	// ====== Axis enable =====	
		bCmdEnableAxis 		: BOOL 	:= FALSE; // Command to enable the axis (External)
		bInternalEnable		: BOOL 	:= FALSE; // internal enable command (turns off after set time, and on at new motion command
		bDelayedEnable		: BOOL 	:= false; // Delayed enable signal for motion commands
		TonMotionEnable		: TON 			; // Timer on for motion command enable
		TofIntAxisEnable	: TOF  			; // Timer off for internal axis enable 
	// ===== Safe commands =====
		bCmdSafeStop	: BOOL ;
	// Motion commands 
		fbMcPower 			: MC_Power		;		// FB for enable and override
		fbMcReset 			: MC_Reset		;		// FB to reset axis
		fbSoeReset			: FB_SoEReset	; 		// FB to reset axis hardware
		fbMcHome			: MC_Home		;		// Fb to home Axis
		fbMcStop 			: MC_Stop		;		// FB to stop axis
		fbMcHalt			: MC_Halt		;		// FB to halt axis
		fbMcJog				: MC_Jog		;		// FB to Jog axis
		fbMcMoveVelocity	: MC_MoveVelocity;		// FB to move with specified velocity until Next command is given
	(* PtoP Motion move commands are in arrays so multiple commands can be stacked *) 
		fbMCMoveRelative	: ARRAY [0..1] OF MC_MoveRelative	;		// FB to move relative
		fbMcMoveAbsolute	: ARRAY [0..1] OF MC_MoveAbsolute	;		// FB to move axis (velocity movement)
		
	// Parameters 
		stMParMaxAcc : Udt_Parameter := (fMaximum := 999999, fMinimum := 0, fValue := 0)	; // Parameter for maximum acceleration
		stMParMaxDec : Udt_Parameter := (fMaximum := 999999, fMinimum := 0, fValue := 0)	; // Parameter for maximum Deceleration
		stMparMaxVelo: Udt_Parameter := (fMaximum := 999999, fMinimum := 0, fValue := 0)	; // Parameter for maximum velocity
		
	// Device feedback
		nActVelocity AT%I* : INT ; // actual speed of the motor
		nActPosition AT%I* : UDINT ; // Actual position of the motor

	// ===== Function execute triggers =====
		bExec_Reset			: BOOL := FALSE; // Execute reset
		bExec_Halt			: BOOL := FALSE; // Execute hold
		bExec_Home			: BOOL := FALSE; // Execute Home
		bExec_JogPositive	: BOOL := FALSE; // Execute Jog in positive direction
		bExec_JogNegative	: BOOL := FALSE; // Execute Jog in negative direction
		bExec_MoveVelocity	: BOOL := FALSE; // Execute move velocity
		arExec_MoveRelative	: ARRAY [0..1] OF BOOL ; // Execute move relative
		arExec_MoveAbs		: ARRAY [0..1] OF BOOL ; // Execute move absolute reverse
		

END_VAR

// Call base function
SUPER^();

// ==== Check if axis is initiated =====
IF NOT bInitOk THEN 
	RETURN ; 
END_IF

// ===== Execute safe functions =====
	ExecSafeFunctions(); 

// ==== Execute organizational functions =====
	ExecEnable();

// ==== execute motion functions =====
	CallMotionFunctions();

METHOD PRIVATE CallMotionFunctions : BOOL
VAR_INPUT
END_VAR
// ===== Check if safe to move =====
	IF bCmdSafeStop OR NOT bDelayedEnable THEN 
		RETURN ;
	END_IF

// ===== Homing functions =====
	ExecHome		(); 

// ===== Motion standstil commands =====
	ExecHalt		();

// ===== Motion move functions
	ExecJog			(); 
	ExecMoveAbsolute();
	ExecMoveRelative();
	ExecMoveVelocity();
END_METHOD

METHOD PUBLIC CmdHalt : BOOL
VAR_INPUT
	fDeceleration 	: LREAL := 0 ; // command deceleration
	mcBuffermode	: MC_BufferMode ; // Buffermode defines how the previous command is executed.
END_VAR
// Set command to true 
bExec_Halt 		:= TRUE ;
bInternalEnable	:= TRUE ;

// copy parameters
fbMcHalt.Deceleration	:= fDeceleration;
fbMcHalt.BufferMode		:= mcBuffermode	;

// Set feedback output 
CmdHalt := fbMchalt.Active ;
END_METHOD

METHOD PUBLIC CmdHome : BOOL // start axis homing procedure
VAR_INPUT
	fPosition 		: LREAL := 0 ; // Homing position
	mcBufferMode	: MC_BufferMode := MC_BufferMode.MC_Aborting		; // Buffermode
END_VAR
// set command to true 
bExec_Home 		:= TRUE	; 
bInternalEnable	:= TRUE ;

// copy parameters
fbMcHome.Position 	:= fPosition 	;
fbMcHome.BufferMode	:= mcBufferMode ;

// Set feedback output
CmdHome := fbMcHome.Done ;
END_METHOD

METHOD PUBLIC CmdJog : BOOL // Jog axis with variable speed. jog stops as soon as the command is false
VAR_INPUT
	fVelocity		: LREAL 	; // jog velocity can be adjusted as long as the command is active
	fPos			: LREAL 	; // Jog position or step size (if aplicable)
	bJogNegative 	: BOOL 		:= FALSE ; // jog in negative direction
	eJogmode		: E_JogMode := E_JogMode.MC_JOGMODE_CONTINOUS ; // jogmode [default MC_JOGMODE_CONTINOUS] 
END_VAR
// Velocity conversion from RPM to deg/sec
	IF bIcfCmdVelocityRpm THEN 
		fVelocity := Rpm_To_DegS(fVelocity);
	END_IF

// Set command to true
	IF fbMcJog.Velocity = fVelocity THEN // If command velocity changes, then set exec to false for one cycle to trigger new velocity so the jog follows the set velocity
		bExec_JogPositive	:= NOT bJogNegative ;
		bExec_JogNegative 	:= bJogNegative ;
	END_IF
	bInternalEnable			:= TRUE ;

// copy parameters
	fbMcJog.Velocity	:= fVelocity 	;
	fbmcjog.Mode		:= eJogmode		;
	fbMcJog.Position	:= fPos			;

// Set feedback output 
	CmdJog := fbMcJog.Active ;
END_METHOD

METHOD PUBLIC CmdManual : BOOL
VAR
	eJogmode		: E_JogMode := E_JogMode.MC_JOGMODE_CONTINOUS ; // jogging mode 
END_VAR
// Enable axis for manual control
bCmdManual := TRUE ;

// set jog mode 
IF stManualCtrl.bCmdInching THEN 
	eJogmode := E_JogMode.MC_JOGMODE_INCHING ;
END_IF

// execute motion commands
IF stManualCtrl.bCmdJogForward OR stManualCtrl.bCmdJogReverse THEN 
	CmdJog (fVelocity := stManualCtrl.fVelocity, 
			fPos := stManualCtrl.fDistance, 
			bJogNegative := stManualCtrl.bCmdJogReverse, 
			eJogmode := eJogmode);
ELSIF stManualCtrl.bCmdToPos THEN 
	CmdMoveAbs( fPosition := stManualCtrl.fPosition, 
				fVelocity := stManualCtrl.fVelocity, 
				mcBuffermode := MC_BufferMode.MC_Aborting);
ELSIF stManualCtrl.bCmdHome THEN 
	CmdHome( fPosition := 0, mcBufferMode := MC_Aborting);
ELSE 
	CmdHalt( 	fDeceleration := fMaxDec * 0.9, 
				mcBuffermode := MC_BufferMode.MC_Aborting) ; 
END_IF
END_METHOD

METHOD PUBLIC CmdMoveAbs : BOOL // Move absolute command
VAR_INPUT
	fPosition	:	LREAL 	; // target position
	fVelocity	: 	LREAL 	; // Maximum velocity [units/sec]
	mcBuffermode: 	MC_BufferMode ; // Buffermode defines how the previous command is executed.
END_VAR
// Velocity conversion from RPM to deg/sec
	IF bIcfCmdVelocityRpm THEN 
		fVelocity := Rpm_To_DegS(fVelocity);
	END_IF

// Determine function for command stacking
	IF fbMcMoveAbsolute[0].Active THEN 
		arExec_MoveAbs[1] 				:= (fPosition <> fbMcMoveAbsolute[0].Position OR fVelocity <> fbMcMoveAbsolute[0].Velocity) ;
		fbMcMoveAbsolute[1].Position 	:= fPosition ;
		fbMcMoveAbsolute[1].Velocity 	:= fVelocity ; 
		fbMcMoveAbsolute[1].BufferMode 	:= mcBuffermode ;
	ELSE
		arExec_MoveAbs[0] 				:= (fPosition <> fbMcMoveAbsolute[1].Position OR fVelocity <> fbMcMoveAbsolute[1].Velocity) ;
		fbMcMoveAbsolute[0].Position 	:= fPosition ;
		fbMcMoveAbsolute[0].Velocity 	:= fVelocity ; 
		fbMcMoveAbsolute[0].BufferMode 	:= mcBuffermode ;
	END_IF

bInternalEnable	:= TRUE ;
// set feedback
IF arExec_MoveAbs[1] OR fbMcMoveAbsolute[1].Busy THEN 
	CmdMoveAbs :=	fbMcMoveAbsolute[1].Active ;
ELSE 
	CmdMoveAbs :=	fbMcMoveAbsolute[0].Active ;
END_IF
END_METHOD

METHOD CmdMoveRelative : BOOL // move relative command 
VAR_INPUT
	fDistance	:	LREAL 	; // target position
	fVelocity	: 	LREAL 	; // Maximum velocity [units/sec]
	mcBuffermode: 	MC_BufferMode ; // Buffermode defines how the previous command is executed.
END_VAR
// Velocity conversion from RPM to deg/sec
	IF bIcfCmdVelocityRpm THEN 
		fVelocity := Rpm_To_DegS(fVelocity);
	END_IF

// Determine function for command stacking
	IF fbMCMoveRelative[0].Active THEN 
		arExec_MoveRelative[1] := (fDistance <> fbMCMoveRelative[0].Distance OR fVelocity <> fbMCMoveRelative[0].Velocity) ;
		fbMCMoveRelative[1].Velocity	:= fVelocity 	;
		fbMCMoveRelative[1].Distance	:= fDistance	;
		fbMCMoveRelative[1].BufferMode	:= mcBuffermode	;
	ELSE 
		arExec_MoveRelative[0] := (fDistance <> fbMCMoveRelative[1].Distance OR fVelocity <> fbMCMoveRelative[1].Velocity) ;
		fbMCMoveRelative[0].Velocity	:= fVelocity 	;
		fbMCMoveRelative[0].Distance	:= fDistance	;
		fbMCMoveRelative[0].BufferMode	:= mcBuffermode	;
	END_IF

bInternalEnable	:= TRUE ;

// set feedback
IF arExec_MoveRelative[1] OR fbMCMoveRelative[1].Busy THEN 
	CmdMoveRelative :=	fbMCMoveRelative[1].Active ;
ELSE
	CmdMoveRelative :=	fbMCMoveRelative[0].Active ;
END_IF
END_METHOD

METHOD PUBLIC CmdMoveVelocity : BOOL // Move with set velocity until stopped
VAR_INPUT
	fVelocity	: 	LREAL 	; // Maximum velocity [units/sec]
	mcDirection : 	MC_Direction := MC_Direction.MC_Positive_Direction ; // Direction of movement mc_direction [ deafult mc_positive_direction]
	mcBuffermode: 	MC_BufferMode ; // Buffermode defines how the previous command is executed.
END_VAR
// Velocity conversion from RPM to deg/sec
	IF bIcfCmdVelocityRpm THEN 
		fVelocity := Rpm_To_DegS(fVelocity);
	END_IF

// Set command to true 
	bExec_MoveVelocity 	:= TRUE ;
	bInternalEnable		:= TRUE ;

// copy parameters
	fbMcMoveVelocity.Velocity	:= fVelocity 	;
	fbMcMoveVelocity.Direction 	:= mcDirection	;
	fbMcMoveVelocity.BufferMode	:= mcBuffermode	;

// Set feedback output 
	CmdMoveVelocity := fbMcMoveVelocity.Active ;
END_METHOD

METHOD PUBLIC CmdReset : BOOL
VAR_INPUT
END_VAR
// Set reset axis to true 				
	bExec_Reset 	:= TRUE ; 
	bInternalEnable	:= TRUE ;
	
// Set feedback output 
	CmdReset := fbMcReset.Done ;
END_METHOD

METHOD PUBLIC CmdSafeStop : BOOL
VAR_INPUT
END_VAR
// Set safestop command
bCmdSafeStop := TRUE ; 

// Set feedback output 
CmdSafeStop := bIsSafe OR NOT bInitOk;
END_METHOD

METHOD PRIVATE ExecEnable : BOOL
VAR_INPUT
END_VAR
// ===== Set axis enable ======
IF NOT bEnable AND NOT bCmdManual AND nActVelocity <> 0 THEN
	CmdHalt(fDeceleration := fCmdDecc, mcBuffermode := MC_BufferMode.MC_Aborting);
ELSE 
	bCmdEnableAxis	:= bEnable OR bCmdManual ;
	bCmdManual := FALSE ;
END_IF

// ===== Check if axis is bussy with a command =====
	bInternalEnable	S= bIcfAlwaysEnable ; // always enable axis if configured
	
// ===== Axis disable timer after last command =====
	TofIntAxisEnable (	IN:= bInternalEnable, PT := tDisableDelay);

// ===== Enable drive =====
	fbMcPower(	Axis			:= AxisRef , 
				Enable			:= bCmdEnableAxis AND TofIntAxisEnable.Q, 
				Enable_Positive	:= bIcfEnableForward, 
				Enable_Negative	:= bIcfEnableReverse, 
				Override		:= 100 );  
				
// ===== Reset internal enable signal =====
	bInternalEnable := FALSE ; 	

// ===== Delayed enable function =====	
	TonMotionEnable(IN := fbMcPower.Active, PT := tEnableDelay);
	bDelayedEnable := TonMotionEnable.Q ;	


IF fbMcPower.Error THEN 
	bErrorActive			:= TRUE							;
	stFault.Active 			:= TRUE 						;
	stFault.Description		:= CONCAT('Enable Fault ', UDINT_TO_STRING(fbMcPower.ErrorID));				;
	stFault.FaultType		:= E_FaultTypes.FF				;
END_IF
END_METHOD

METHOD PRIVATE ExecHalt : BOOL
VAR_INPUT
END_VAR
// ==== Execute halt function ===== 
fbMcHalt (	Axis 		:= AxisRef,
			Execute 	:= bExec_Halt );

// ===== reset command =====
	bExec_Halt := FALSE ;
	bInternalEnable := fbMcHalt.Busy ;			
	
// Halt fault handling 
	IF fbMcHalt.Error THEN 
		bErrorActive			:= TRUE							;
		stFault.Active 			:= TRUE 						;
		stFault.Description		:= CONCAT('Halt Fault ', UDINT_TO_STRING(fbMcHalt.ErrorID));				;
		stFault.FaultType		:= E_FaultTypes.FF				;
	END_IF
END_METHOD

METHOD PRIVATE ExecHome : BOOL
VAR_INPUT
END_VAR
// ==== execute homing function =====
	fbMcHome(	Axis			:= AxisRef,
				Execute			:= bExec_Home,
				HomingMode		:= MC_DefaultHoming ); 
			
// Reset exec command 
	bExec_Home 	:= FALSE ;
	bHomed		S= fbMcHome.Done ;	
	bInternalEnable := fbMcHome.Busy ;			
				
// fault handling 
	IF fbMcHome.Error THEN 
		bErrorActive			:= TRUE							;
		stFault.Active 			:= TRUE 						;
		stFault.Description		:= CONCAT('Homing Fault ', UDINT_TO_STRING(fbMcHome.ErrorID));				;
		stFault.FaultType		:= E_FaultTypes.FF				;
	END_IF
END_METHOD

METHOD PRIVATE ExecJog : BOOL
VAR_INPUT
END_VAR
// ===== Execute Jog function =====
	// function call
	fbMcJog (	Axis 		:= AxisRef,
				JogForward	:= bExec_JogPositive,
				JogBackwards:= bExec_JogNegative,
				Acceleration:= fCmdAcc,
				Deceleration:= fCmdDecc );

// ===== reset command =====
	bExec_JogPositive 	:= FALSE  ;
	bExec_JogNegative	:= FALSE  ;
	bInternalEnable		:= fbMcJog.Busy; 

// Jog fault handling 
	IF fbMcJog.Error THEN 
		bErrorActive			:= TRUE							;
		stFault.Active 			:= TRUE 						;
		stFault.Description		:= CONCAT('Jog Fault ', UDINT_TO_STRING(fbMcJog.ErrorID));				;
		stFault.FaultType		:= E_FaultTypes.FF				;
	END_IF
END_METHOD

METHOD PRIVATE ExecMoveAbsolute : BOOL
VAR_INPUT
END_VAR
VAR
	i : UDINT := 0 ;
END_VAR
// ==== execute move absolute function =====
FOR i := 0 TO 1 DO 
	// function call
	fbMcMoveAbsolute[i](	Axis 		:= AxisRef,
							Execute 	:= arExec_MoveAbs[i],
							Acceleration:= fCmdAcc,
							Deceleration:= fCmdDecc );  
	// reset Exec command 
	arExec_MoveAbs[i] := FALSE ; 
	bInternalEnable := fbMcMoveAbsolute[i].Busy ;			

	// If function is done then reset command values
	IF fbMcMoveAbsolute[i].Done THEN 
		fbMcMoveAbsolute[i].Velocity	:= 0 ;
		fbMcMoveAbsolute[i].Position	:= 0 ; 
	END_IF
	
	// fault handling 
	IF fbMcMoveAbsolute[i].Error THEN 
		bErrorActive			:= TRUE							;
		stFault.Active 			:= TRUE 						;
		stFault.Description		:= CONCAT('Move absolute Fault ', UDINT_TO_STRING(fbMcMoveAbsolute[i].ErrorID));				;
		stFault.FaultType		:= E_FaultTypes.FF				;
	END_IF
END_FOR
END_METHOD

METHOD PRIVATE ExecMoveRelative : BOOL
VAR_INPUT
END_VAR
VAR
	i : UDINT := 0 ;
END_VAR
// ===== Execute move relative function ======
FOR i := 0 TO 1 DO 
	// function call
	fbMCMoveRelative[i](	Axis 		:= AxisRef,
							Execute		:= arExec_MoveRelative[i],
							Acceleration:= fCmdAcc,
							Deceleration:= fCmdDecc );
	// reset Exec command 
	arExec_MoveRelative[i] := FALSE ; 
	bInternalEnable := fbMCMoveRelative[i].Busy ;			

	// If function is done then reset command values
	IF fbMCMoveRelative[i].Done THEN 
		fbMCMoveRelative[i].Velocity	:= 0 ;
		fbMCMoveRelative[i].Distance	:= 0 ; 
	END_IF
	
	// fault handling 
	IF fbMCMoveRelative[i].Error THEN 
		bErrorActive			:= TRUE							;
		stFault.Active 			:= TRUE 						;
		stFault.Description		:= CONCAT('Move relative Fault ', UDINT_TO_STRING(fbMCMoveRelative[i].ErrorID));				;
		stFault.FaultType		:= E_FaultTypes.FF			;
	END_IF
END_FOR
END_METHOD

METHOD PRIVATE ExecMoveVelocity : BOOL
VAR_INPUT
END_VAR
// ===== Execute move velocity function =====
// function call
fbMcMoveVelocity (	Axis 		:= AxisRef,
					Execute		:= bExec_MoveVelocity,
					Acceleration:= fCmdAcc,
					Deceleration:= fCmdDecc );

// ===== reset command =====
bExec_MoveVelocity := FALSE ;
bInternalEnable		:= fbMcMoveVelocity.Busy;
	
// Halt fault handling 
IF fbMcHalt.Error THEN 
	bErrorActive			:= TRUE							;
	stFault.Active 			:= TRUE 						;
	stFault.Description		:= CONCAT('Move velocity Fault ', UDINT_TO_STRING(fbMcMoveVelocity.ErrorID));				;
	stFault.FaultType		:= E_FaultTypes.FF				;
END_IF
END_METHOD

METHOD PRIVATE ExecReset : BOOL
VAR_INPUT
END_VAR
IF  nActVelocity <> 0 AND bExec_Reset THEN // If the axis is still moving execute safe stop first
	CmdSafeStop();
	RETURN;
END_IF

// perform reset 
	fbMcReset	( 	Execute	:= bexec_reset AND NOT fbSoeReset.Busy,
					Axis	:= AxisRef ); 
					
// ===== reset command =====
	bExec_Reset := FALSE ;
	
// ===== reset internal fault bits and stop bits =====
	bErrorActive 			:= FALSE ; 
	
// ===== reset safe commands ======
	bCmdSafeStop	:= FALSE ; 
	
// Reset fault handling 
	IF fbSoeReset.Error OR fbMcReset.Error THEN 
		bErrorActive			:= TRUE							;
		stFault.Active 			:= TRUE 						;
		stFault.Description		:= CONCAT('Reset Fault ', UDINT_TO_STRING(fbMcReset.ErrorID))			;
		stFault.FaultType		:= E_FaultTypes.FF				;
	END_IF
END_METHOD

METHOD PRIVATE ExecSafeFunctions : BOOL
VAR_INPUT
END_VAR
// ==== Safe operation functions (overrule all other motion functions) =====
	fbMcStop( 	Axis 			:= AxisRef		,
				Execute 		:= bCmdSafeStop	,
				Deceleration	:= fMaxDec		);
	
	// Reset axis command			
	bCmdSafeStop 	R= fbMcStop.Done ;
	
// Safestop fault handling 
	IF fbMcStop.Error THEN 
		bErrorActive			:= TRUE							;
		stFault.Active 			:= TRUE 						;
		stFault.Description		:= CONCAT('Safe stop axis fault ', UDINT_TO_STRING(fbMcStop.ErrorID));				;
		stFault.FaultType		:= E_FaultTypes.FF				;
	END_IF

// ===== Dev is safe feedback =====
bIsSafe := NOT bCmdEnableAxis  ;
END_METHOD

METHOD PUBLIC Init : BOOL
VAR_INPUT
	// Message location data
	nId			: UINT ; // Identification number of object
	nParentId	: UDINT ; // Id of higher level If aplicable (0 = no parent)
	// Config Bits
	bIcfCmdVelocityRpm	: BOOL := FALSE ; // input speeds in Rpm
	bIcfEnableForward 	: BOOL := TRUE 	; // Enable forward motion
	bIcfEnableReverse	: BOOL := TRUE 	; // Enable reverse motion
	bIcfAlwaysEnable	: BOOL := FALSE ; // 1 = Axis always enabled, 0 = Axis disabled at Idle 
	bIcfSimulationMode	: BOOL := FALSE ; // Simulation mode is active [default set to False] Used for testing without hardware present 
	
	fHomePosition		: LREAL := 0 	; // set position at homing
	fSafeVeloLimit		: LREAL	:= 360 	; // safe velocity limit [deg/sec]
	nEncTurnoverVal 	: LREAL := 360	; // encoder turnover value 
	tEnableDelay		: time 	:= T#0MS; // Time between axis enable command and motion command execution (0 := no delay active)	
	tDisabledelay		: TIME 	:= T#100MS; // Axis idle time before axis is disabled 
END_VAR
VAR 
	bActParamValid 		: BOOL ; // Parameter read is valid 
END_VAR
// ====== Set init to true =====
	bInitOk	:= TRUE ; 

// ====== Calculate device id =====
	bInitOk :=	ExecIdentifyDevice(nId,nParentId, E_ComponentTypes.Axis) AND bInitOk;

// ===== Write parameters =====
	stMParMaxAcc.nNumber		:= stIdentity.nLocationId + 1;
	stMParMaxAcc.sDiscription 	:= CONCAT(STR1 := stIdentity.sName, STR2:= ' hardware maximum acceleration (0 = HWMaximum)'); 
	stMParMaxAcc.sName			:= CONCAT(STR1 := stIdentity.sName, STR2:= ' Hard max acceleration');
	stMParMaxAcc.sType			:= 'MPar';
	stMParMaxAcc.sUnit			:= 'unit/s^2';
	
	stMParMaxDec.nNumber		:= stIdentity.nLocationId + 2;
	stMParMaxDec.sDiscription 	:= CONCAT(STR1 := stIdentity.sName, STR2:= ' hardware maximum deceleration(0 = HWMaximum)'); 
	stMParMaxDec.sName			:= CONCAT(STR1 := stIdentity.sName, STR2:= ' Hard max deceleration');
	stMParMaxDec.sType			:= 'MPar';
	stMParMaxDec.sUnit			:= 'unit/s^2';
	
	stMparMaxVelo.nNumber		:= stIdentity.nLocationId + 3;
	stMparMaxVelo.sDiscription 	:= CONCAT(STR1 := stIdentity.sName, STR2:= ' hardware maximum velocity'); 
	stMparMaxVelo.sName			:= CONCAT(STR1 := stIdentity.sName, STR2:= ' Hard max velocity');
	stMparMaxVelo.sType			:= 'MPar';
	stMparMaxVelo.sUnit			:= 'Units/s';

	refFbParHandler.CmdAddParameter(refParameter := stMParMaxAcc);
	refFbParHandler.CmdAddParameter(refParameter := stMParMaxDec);
	refFbParHandler.CmdAddParameter(refParameter := stMparMaxVelo);

// ===== set axis configuration =====	
	fMaxAcc	:= stMParMaxAcc.fValue;
	fMaxDec	:= stMParMaxDec.fValue;	
	fMaxVelo:= stMparMaxVelo.fValue;

	fCmdAcc 		:= fMaxAcc;
	fCmdDecc		:= fMaxDec;
// ===== Configure Axis =====
	// ***** Config Bits *****
		THIS^.bIcfCmdVelocityRpm	:= bIcfCmdVelocityRpm	; // Enable speed inputs in Rpm
		THIS^.bIcfEnableForward 	:= bIcfEnableForward 	; // Enable forward motion
		THIS^.bIcfEnableReverse		:= bIcfEnableReverse	; // Enable reverse motion
		THIS^.bIcfAlwaysEnable		:= bIcfAlwaysEnable		; // Always enable motor and brake if safety is ok
		THIS^.bIcfSimulationMode	:= bIcfSimulationMode 	; // Simulation mode is active [default set to False] 

	// ***** config homing Mode ***** 
 		THIS^.fHomePosition			:= fHomePosition;
	// ***** Velocity settings *****
		THIS^.fSafeVeloLimit 		:= fSafeVeloLimit ; // set maximum safe velocity	
	// ***** Time delay enable off *****
		THIS^.tEnableDelay		:= tEnableDelay	;
		THIS^.tDisableDelay 	:= tDisabledelay ;		

// ===== Set device type for manual control =====
	eDevType := E_Devices.Axis ;
		
// ===== reset axis state indicators ======
	bErrorActive 	:= FALSE;
END_METHOD

END_FUNCTION_BLOCK

// ---- Axis/FunctionBlocks/ServoHybrid/FB_DevHybridAc.TcPOU
{attribute 'reflection'}
FUNCTION_BLOCK PUBLIC FB_DevHybridAc EXTENDS Fb_DevAxis
VAR_INPUT
END_VAR
VAR_OUTPUT
END_VAR
VAR
	// Parameters 
		stMParMaxAcc : Udt_Parameter := (fMaximum := 999999, fMinimum := 0, fValue := 0)	; // Parameter for maximum acceleration
		stMParMaxDec : Udt_Parameter := (fMaximum := 999999, fMinimum := 0, fValue := 0)	; // Parameter for maximum Deceleration
		stMparMaxVelo: Udt_Parameter := (fMaximum := 999999, fMinimum := 0, fValue := 0)	; // Parameter for maximum velocity
END_VAR

SUPER^();

METHOD INTERNAL ExecHalt : BOOL
VAR_INPUT
END_VAR
// The hybrid axis is equiped with it's own safety stop system therefore mc halt is no longer needed with an Estop

// ==== Execute halt function ===== 
fbMcHalt (	Axis 		:= AxisRef,
			Execute 	:= bExec_Halt );

// ===== reset command =====
	bExec_Halt := FALSE ;
	
// Halt fault handling 
	IF fbMcHalt.Error THEN 
		bError					:= TRUE							;
		stFault.Active 			:= TRUE 						;
		stFault.Description		:= CONCAT('Halt Fault ', UDINT_TO_STRING(fbMcHalt.ErrorID));				;
		stFault.FaultType		:= E_FaultTypes.FF				;
	END_IF
END_METHOD

METHOD INTERNAL ExecReadStatus : BOOL
VAR_INPUT
END_VAR
// Read axis status from drive
AxisRef.ReadStatus();						
// convert velocity to RPM for output if aplicable
IF bIcfCmdVelocityRpm THEN 
	fVelocity := AxisRef.NcToPlc.ActVelo / 6 ;
ELSE 
	fVelocity := AxisRef.NcToPlc.ActVelo ;
END_IF

// write position output
fActPosition := AxisRef.NcToPlc.ActPos ;
						
// set status bits 
bIdle := NOT AxisRef.Status.HasJob ;
END_METHOD

METHOD INTERNAL ExecReset : BOOL
VAR_INPUT
END_VAR
IF  AxisRef.Status.Moving AND bExec_Reset THEN // If the axis is still moving execute safe stop first
	CmdSafeStop();
	RETURN;
END_IF

	fbMcReset	( 	Execute	:= bexec_reset,
					Axis	:= AxisRef ); 
					
// ===== reset command =====
	bExec_Reset := FALSE ;
	
// ===== reset internal fault bits and stop bits =====
	bError 			:= FALSE ; 
	
// ===== reset safe commands ======
	bCmdSafeStop	:= FALSE ; 
	bCmdSafeSpeed 	:= FALSE ;
	
// Reset fault handling 
	IF fbMcReset.Error THEN 
		bError					:= TRUE							;
		stFault.Active 			:= TRUE 						;
		stFault.Description		:= CONCAT('Reset Fault ', UDINT_TO_STRING(fbMcReset.ErrorID))			;
		stFault.FaultType		:= E_FaultTypes.FF				;
	END_IF
END_METHOD

METHOD PUBLIC Init : BOOL
VAR_INPUT
	// Message location data
	nId			: UINT ; // Identification number of object
	nParentId	: UDINT ; // Id of higher level If aplicable (0 = no parent)
	// Config Bits
	bIcfCmdVelocityRpm	: BOOL := FALSE ; // input speeds in Rpm
	bIcfEnableForward 	: BOOL := TRUE 	; // Enable forward motion
	bIcfEnableReverse	: BOOL := TRUE 	; // Enable reverse motion
	bIcfAlwaysEnable	: BOOL := FALSE ; // 1 = Axis always enabled, 0 = Axis disabled at Idle 
	bIcfModuloAxis		: BOOL := FALSE ; // Show axis position as modulo
	bIcfSTOPresent		: BOOL := FALSE ; // Axis safe torque off is present	
	bIcfNCHomeSensor	: BOOL := FALSE ; // Homing sensor is inverted (NC)	

	// Config Values 
	mcHomingMode 		: MC_HomingMode := MC_HomingMode.MC_DefaultHoming; 
	fSafeOverride		: LREAL := 10	; // Safe velocity override [%]
	nEncTurnoverVal 	: LREAL := 360	; // encoder turnover value 
	tEnableDelay		: time 	:= T#0MS; // Time between axis enable command and motion command execution (0 := no delay active)	
	tDisabledelay		: TIME 	:= T#100MS; // Axis idle time before axis is disabled 
END_VAR
VAR 
	bActVeloReadValid 	: BOOL ; // velocity parameter read is valid 
	bActAccReadValid 	: BOOL ; // Acceleration parameter read is valid 
	bActDecReadValid 	: BOOL ; // Deceleration parameter read is valid 
	bActParamValid 		: BOOL ; // Parameter read is valid 
END_VAR
// Calculate device number
	ExecIdentifyDevice(nId,nParentId, E_ComponentTypes.Axis);

// ===== Write parameters =====
	stMParMaxAcc.nNumber		:= stIdentity.nLocationId + 1;
	stMParMaxAcc.sDiscription 	:= CONCAT(STR1 := stIdentity.sName, STR2:= ' hardware maximum acceleration (0 = HWMaximum)'); 
	stMParMaxAcc.sName			:= CONCAT(STR1 := stIdentity.sName, STR2:= ' Hard max acceleration');
	stMParMaxAcc.sType			:= 'MPar';
	stMParMaxAcc.sUnit			:= 'unit/s^2';
	
	stMParMaxDec.nNumber		:= stIdentity.nLocationId + 2;
	stMParMaxDec.sDiscription 	:= CONCAT(STR1 := stIdentity.sName, STR2:= ' hardware maximum deceleration(0 = HWMaximum)'); 
	stMParMaxDec.sName			:= CONCAT(STR1 := stIdentity.sName, STR2:= ' Hard max deceleration');
	stMParMaxDec.sType			:= 'MPar';
	stMParMaxDec.sUnit			:= 'unit/s^2';
	
	stMparMaxVelo.nNumber		:= stIdentity.nLocationId + 3;
	stMparMaxVelo.sDiscription 	:= CONCAT(STR1 := stIdentity.sName, STR2:= ' hardware maximum velocity'); 
	stMparMaxVelo.sName			:= CONCAT(STR1 := stIdentity.sName, STR2:= ' Hard max velocity');
	stMparMaxVelo.sType			:= 'MPar';
	stMparMaxVelo.sUnit			:= 'Units/s';

	refFbParHandler.CmdAddParameter(refParameter := stMParMaxAcc);
	refFbParHandler.CmdAddParameter(refParameter := stMParMaxDec);
	refFbParHandler.CmdAddParameter(refParameter := stMparMaxVelo);

// ===== set axis configuration =====	
	fMaxAcc	:= stMParMaxAcc.fValue;
	fMaxDec	:= stMParMaxDec.fValue;	
	fMaxVelo:= stMparMaxVelo.fValue;

	fCmdAcc 		:= fMaxAcc;
	fCmdDec		:= fMaxDec;
// ===== Configure Axis =====
	// ***** Config Bits *****
		THIS^.bIcfCmdVelocityRpm	:= bIcfCmdVelocityRpm	; // Enable speed inputs in Rpm
		THIS^.bIcfEnableForward 	:= bIcfEnableForward 	; // Enable forward motion
		THIS^.bIcfEnableReverse		:= bIcfEnableReverse	; // Enable reverse motion
		THIS^.bIcfAlwaysEnable		:= bIcfAlwaysEnable		; // Always enable motor and brake if safety is ok

	// ***** config homing Mode ***** 
 		THIS^.mcHomingMode 			:= mcHomingMode ; // set homing mode
	// ***** Velocity settings *****
		THIS^.fSafeOverride			:= fSafeOverride	; 	
	// ***** Time delay enable off *****
		THIS^.tEnableDelay		:= tEnableDelay	;
		THIS^.tDisableDelay 	:= tDisabledelay ;		

// ===== Set device type for manual control =====
	eDevType := E_Devices.Axis ;
		
// ===== reset axis state indicators ======
	bErrorActive 	:= FALSE;

// ====== Set init to done =======
	bInitOk	:= TRUE ;
END_METHOD

END_FUNCTION_BLOCK

// ---- Axis/FunctionBlocks/TwoVelocityControl/FB_DevTwoVelocityAxis.TcPOU
{attribute 'reflection'}
FUNCTION_BLOCK PUBLIC FB_DevTwoVelocityAxis EXTENDS FB_DevBase IMPLEMENTS iTwoDirectionalMotorWithFast
VAR // internal commands
	bCmdRunCW		: BOOL ; // run clockwise
	bCmdRunCWFast	: BOOL ; // Run fast
	bCmdRunCCW		: BOOL ; // run counter clockwise
	bCmdRunCCWFast	: BOOL ; // Run fast
	stManualControl	: st_ManualDigitalMotorControl ; // Manual control structure
END_VAR
VAR // Outputs
	qbRunCw			AT%Q* : BOOL ; // Output run clockwise
	qbRunCWFast		AT%Q* : BOOL ; // Output run clockwise Fast
	qbRunCCW 		AT%Q* : BOOL ; // Output run counter clockwise
	qbRunCCWFast	AT%Q* : BOOL ; // Output run Counter clockwise Fast	
END_VAR

SUPER^();

IF NOT bInitOk THEN
	RETURN;
END_IF

ExecSetOutputs();

METHOD PUBLIC CmdManual : BOOL
bCmdManual S= TRUE;

CmdManual := TRUE ;
END_METHOD

METHOD CmdRunCCW : BOOL
bCmdRunCCW := TRUE;

CmdRunCCW := qbRunCCW;
END_METHOD

METHOD CmdRunCCWFast : BOOL
bCmdRunCCWFast := TRUE;

CmdRunCCWFast := qbRunCCWFast;
END_METHOD

METHOD CmdRunCW : BOOL
bCmdRunCW := TRUE;

CmdRunCW := qbRunCW;
END_METHOD

METHOD CmdRunCWFast : BOOL
bCmdRunCWFast := TRUE;

CmdRunCWFast := qbRunCWFast;
END_METHOD

METHOD PUBLIC CmdSafeStop : BOOL
VAR_INPUT
END_VAR
bIsSafe := TRUE;

bIsSafe R= qbRunCw;
bIsSafe R= qbRunCWFast;
bIsSafe R= qbRunCCW;
bIsSafe R= qbRunCCWFast;	

qbRunCw			:= FALSE;
qbRunCWFast		:= FALSE;
qbRunCCW 		:= FALSE;
qbRunCCWFast	:= FALSE;	

CmdSafeStop := bIsSafe;
END_METHOD

METHOD INTERNAL ExecSetOutputs : BOOL
IF bManual THEN
	qbRunCw			:= stManualControl.bManRunCW;
	qbRunCWFast		:= stManualControl.bManRunCWFast;
	qbRunCCW 		:= stManualControl.bManRunCCw;
	qbRunCCWFast	:= stManualControl.bManRunCCWFast;
ELSIF bEnable THEN
	qbRunCw			:= bCmdRunCW;
	qbRunCWFast		:= bCmdRunCWFast;
	qbRunCCW 		:= bCmdRunCCW;
	qbRunCCWFast	:= bCmdRunCCWFast;
ELSE
	qbRunCw			:= FALSE;
	qbRunCWFast		:= FALSE;
	qbRunCCW 		:= FALSE;
	qbRunCCWFast	:= FALSE;	
END_IF

// reset all commands
bCmdRunCW		:= FALSE;
bCmdRunCWFast	:= FALSE;
bCmdRunCCW		:= FALSE;
bCmdRunCCWFast	:= FALSE;
stManualControl.bManRunCW 		:= FALSE;
stManualControl.bManRunCWFast 	:= FALSE;
stManualControl.bManRunCCw 		:= FALSE;
stManualControl.bManRunCCWFast	:= FALSE;

bCmdManual := FALSE;
END_METHOD

METHOD Init : BOOL
VAR_INPUT
	nId			: UINT ; // Identification number of object
	nParentId	: UDINT ; // Id of higher level If aplicable (0 = no parent)
END_VAR
bInitOk := ExecIdentifyDevice(nId, nParentId, eComponentType := E_ComponentTypes.Axis);

// ===== Set device type for manual control =====
eDevType := E_Devices.TwoVelocityAxis ;

Init := bInitOk;
END_METHOD

END_FUNCTION_BLOCK

// ---- Buttons/Functions/FB_DevHMIButton.TcPOU
{attribute 'reflection'}
FUNCTION_BLOCK PUBLIC FB_DevHMIButton EXTENDS FB_DevBase // Button function for HMI 
VAR_INPUT
	Istatus			: BOOL	:= FALSE;// Digital sensor, Direct input status
	tDelay			: TIME 	:= T#5S	;// Time before delayed signal becomes active 
END_VAR
VAR_OUTPUT
	bFcoInputActive		: BOOL 			;// Digital sensor, Button active state
	bFcoDelay			: BOOL			;// Button, Delayed input status (3 seconds) 
	bFeStatus			: BOOL			;// Button, Falling edge of input signal	
	bReStatus			: BOOL			;// Button, Rising edge of input signal
	TetInputActive		: TIME			;// Button, Time elapsed while button is active
	bInvisible			: BOOL 			;// Button, Button is made invisible
	bDeactivate			: BOOL 			;// Button, Deactivate button 
END_VAR
VAR
	FB_delIStatus	: TON; // Timer function for delayed input status 
	FB_feIStatus	: F_TRIG; // generate falling edge pulse edge from Istatus
	FB_reIStatus	: R_TRIG; // generate falling edge pulse edge from Istatus
END_VAR

// Call base function
SUPER^();

// ***** Direct input when enabled *****
IF bEnable THEN 
	bFcoInputActive := Istatus ;
ELSE 
	bFcoInputActive := FALSE ;
END_IF

// ===== check if function is enabled =====
	IF NOT bEnable THEN 
		bInvisible 	:= TRUE ;
		bDeactivate	:= TRUE ;
		bFcoDelay	:= FALSE;
		RETURN;
	ELSE  
		bInvisible 	:= FALSE ;
		bDeactivate	:= FALSE ;
	END_IF

// ====== process functions if enabled ======
	// ***** Set Delayed inputs and time elapsed ****
		FB_delIStatus(	IN:= bFcoInputActive,
						PT:= tDelay , 
						Q=> bFcoDelay , 
						ET=> TetInputActive 
					  ); // Generate delayed input status from push button input status
	// ***** Edge triggers *****
		FB_feIStatus(CLK:= Istatus , Q=> bFeStatus ); // generate falling edge pulse on pushbutton input
		FB_reIStatus (Clk := Istatus , Q => bReStatus); // Generate rising edge from push button input signal

END_FUNCTION_BLOCK

// ---- Buttons/Functions/FB_DevPushbuttonLight.TcPOU
{attribute 'reflection'}
FUNCTION_BLOCK PUBLIC FB_DevPushbuttonLight EXTENDS Fb_DevDigitalInputFunctions
VAR_OUTPUT
END_VAR
VAR
	fbLight : Fb_DevLight ; // light control 
END_VAR

// Set device type
IF eDevType = E_Devices.Undefined THEN 
	eDevType := E_Devices.PushButtonLight ;
END_IF

SUPER^();

// Light commands
	
fbLight(bEnable := bEnable);

METHOD PUBLIC CmdBlinkFast : BOOL
VAR_INPUT
END_VAR
CmdBlinkFast := fbLight.CmdBlinkFast();
END_METHOD

METHOD PUBLIC CmdBlinkSlow : BOOL
VAR_INPUT
END_VAR
CmdBlinkSlow	:= fbLight.CmdBlinkSlow();
END_METHOD

METHOD PUBLIC CmdOn : BOOL
VAR_INPUT
END_VAR
CmdOn := fbLight.CmdOn() ;
END_METHOD

END_FUNCTION_BLOCK

// ---- Lights/Functions/Fb_DevLight.TcPOU
{attribute 'reflection'}
FUNCTION_BLOCK PUBLIC Fb_DevLight EXTENDS FB_DevBase ;
VAR_OUTPUT
	bSoftLightOut	: BOOL ; // Software light output	
END_VAR
VAR
	bCmdBlinkSlow	: BOOL := FALSE ; // Command light blink slow
	bCmdBlinkFast 	: BOOL := FALSE ; // Command light blink fast
	bCmdOn			: BOOL := FALSE ; // Command turn light on	 
	qLight AT %Q* 	: BOOL := FALSE ; // light output
END_VAR

// set device type
IF eDevType = E_Devices.Undefined THEN 
	eDevType := E_Devices.DigitalOut ;
END_IF

// ===== check if light is enabled ======
	IF NOT bEnable AND NOT bCmdManual THEN 
		qLight := FALSE ;
		RETURN; 
	END_IF
	
// ===== set light output ======
	ExecSetOutput();

METHOD PUBLIC CmdBlinkFast : BOOL
VAR_INPUT
END_VAR
bCmdBlinkFast S= TRUE ;

CmdBlinkFast := bCmdBlinkFast ;
END_METHOD

METHOD PUBLIC CmdBlinkSlow : BOOL
VAR_INPUT
END_VAR
bCmdBlinkSlow S= TRUE ;

CmdBlinkSlow	:= bCmdBlinkSlow ;
END_METHOD

METHOD PUBLIC CmdOn : BOOL
VAR_INPUT
END_VAR
bCmdOn S= TRUE ;

CmdOn := qLight ;
END_METHOD

METHOD PRIVATE ExecSetOutput : BOOL
VAR_INPUT
END_VAR
// ===== set light output state =====
IF bCmdOn THEN 
	qLight S= TRUE ;
ELSIF bCmdBlinkFast THEN 
	qLight := Sys_Variables.BlinkFast 	;
ELSIF bCmdBlinkSlow THEN 
	qLight := Sys_Variables.BlinkSlow	;
ELSE
	qLight := FALSE ;
END_IF

// set soft output
bSoftLightOut	:= qLight;

// reset all commands 
bCmdOn			:= FALSE ;
bCmdBlinkFast 	:= FALSE ;
bCmdBlinkSlow 	:= FALSE ;
END_METHOD

METHOD PUBLIC Init : BOOL
VAR_INPUT
	// Location data for messages  
	nId			: UINT ; // Identification number of object
	nParentId	: UDINT ; // Id of higher level If aplicable (0 = no parent)
END_VAR
// ====== Set init to true =====
	bInitOk	:= TRUE ; 

// ====== Calculate device id =====
	bInitOk :=	ExecIdentifyDevice(nId,nParentId, E_ComponentTypes.DiOutput) AND bInitOk;

// ===== Set feedback =====
	Init := bInitOk;
END_METHOD

END_FUNCTION_BLOCK

// ---- Buttons/Functions/FB_DevPushButton.TcPOU
{attribute 'reflection'}
FUNCTION_BLOCK PUBLIC FB_DevPushButton EXTENDS Fb_DevDigitalInputFunctions
VAR_INPUT
END_VAR
VAR_OUTPUT
END_VAR
VAR
END_VAR

// set device type
IF eDevType = E_Devices.Undefined THEN 
	eDevType := E_Devices.DigitalSensor ;
END_IF

SUPER^();

END_FUNCTION_BLOCK

// ---- CounterCards/FunctionBlocks/KL5151/FB_DevKL5151.TcPOU
{attribute 'reflection'}
FUNCTION_BLOCK FB_DevKL5151 EXTENDS FB_DevBase IMPLEMENTS iCounter
VAR_INPUT
	bInitAsCounterCard	: BOOL := FALSE; // (Default = FALSE) Use Terminal as encoder input (FALSE) or counter (TRUE) 
END_VAR
VAR CONSTANT // register values 
	WRITE_FEATURE_REGISTER 	: USINT := 16#E0; // write to register address command
	READ_FEATURE_REGISTER	: USINT := 16#A0; // Read feature register response  
END_VAR
VAR // Inputs and outputs
	Status		AT%I* : USINT ; // status byte from card
	Counter		AT%I* : UDINT ; // 
	Ctrl 		AT%Q* : USINT ; // Control byte to card`
	DataOut 	AT%Q* : UDINT ; // Set counter value
END_VAR
VAR // steppers
	InitStep : INT := 0; // init stepper
END_VAR
VAR // Manual control
	stManualControl : st_ManualCounterControl;
END_VAR

SUPER^();

METHOD PUBLIC CmdManual : BOOL
bCmdManual := TRUE;
stManualControl.nCount := Counter;

IF stManualControl.bManSetValue THEN 
	// set counter to value
	DataOut	:= stManualControl.nManValue	;
	Ctrl.2 	:= Counter <> stManualControl.nManValue;
	
	stManualControl.bManSetValue R= Counter = stManualControl.nManValue;
END_IF
END_METHOD

METHOD CmdReset : BOOL
VAR_INPUT
END_VAR
Ctrl.2 	:= FALSE;

CmdReset := NOT Status.2;
END_METHOD

METHOD CmdResetValue : BOOL // Reset the value of the counter card to 0
// set counter value to 0
DataOut	:= 0	;
Ctrl.2 	:= Counter <> 0;

CmdResetValue := Counter = 0;
END_METHOD

METHOD PUBLIC CmdSetValue : BOOL // Set the value of the counter card
VAR_INPUT
	Value	: UDINT;
END_VAR
// set counter to value
DataOut	:= Value	;
Ctrl.2 	:= Counter <> Value;

CmdSetValue := Counter = Value;
END_METHOD

PROPERTY PUBLIC CountValue : UDINT
GET
CountValue := Counter;
END_GET
END_PROPERTY

METHOD PUBLIC Init : BOOL
VAR_INPUT
	// Message location data
	nId				: UINT ; // Identification number of object
	nParentId		: UDINT ; // Id of higher level If aplicable (0 = no parent)
END_VAR

IF bInitAsCounterCard THEN
//	{warning 'Counter function needs to be added to devices'}
	ExecIdentifyDevice(nId := nId, nParentId := nParentId, eComponentType := E_ComponentTypes.NA);
ELSE 
	ExecIdentifyDevice(nId := nId, nParentId := nParentId, eComponentType := E_ComponentTypes.Encoder);
END_IF

eDevType := E_Devices.KL5151;

// Check feature register against set function 
CASE InitStep OF 
	0: // check active feature register values
		Ctrl := READ_FEATURE_REGISTER;
		InitStep := initstep + 1;
	1: // Check if operation mode is correct If not set operation mode
		IF Status = READ_FEATURE_REGISTER THEN
			//Check if we are the requested mode
			IF Counter.15 = bInitAsCounterCard THEN 
				InitStep := 3;
			ELSE
				//Copy the current value into the output
				DataOut := Counter;
				//Set the encoder/counter bit as requested
				DataOut.15 := bInitAsCounterCard;
				//Give the command to write to the card
				Ctrl := WRITE_FEATURE_REGISTER;
				InitStep := 2;
			END_IF
		END_IF
	2: // Check if register was written	
		IF Status = READ_FEATURE_REGISTER THEN
			InitStep := 3;
		END_IF
		
	3: //Stop register access, return to normal
		//Copy the current value into the output
		Ctrl := Status;
		//Reset the register access bit
		Ctrl.7 := FALSE;
		InitStep := 4;
		
	4: //Check if the command was accepted
		IF Status.7 = 0 THEN
			InitStep := 10;
		END_IF
		
	10: // init done
		bInitOk := TRUE;
		
	ELSE
		;
END_CASE

Init := bInitOk;
END_METHOD

END_FUNCTION_BLOCK

// ---- Encoders/FunctionBlocks/FB_EncoderBase.TcPOU
{attribute 'reflection'}
FUNCTION_BLOCK PUBLIC FB_EncoderBase EXTENDS FB_DevBase
VAR_OUTPUT
	{attribute 'analysis' := '-33'} // Disable "Unused Variable" rule
	nOutPosition		: LREAL	:= 0	; // Scaled position output
	{attribute 'analysis' := '-33'} // Disable "Unused Variable" rule
	nOutRaw				: UDINT := 0	; // Raw output value	 
	{attribute 'analysis' := '-33'} // Disable "Unused Variable" rule
	nVelocity			: LREAL	:= 0 	; // Velocity [units/sec]
END_VAR
VAR
	fPulsesPerUnit		: LREAL := 1	; // Scale factor for output [units/pulse]
	fOffset				: LREAL := 0	; // Offset for output
	bIcfInverted		: BOOL	:= FALSE; // Invert output position = standard false  
END_VAR

METHOD PUBLIC FastTask : BOOL
VAR_INPUT
END_VAR
END_METHOD

METHOD PUBLIC Init : BOOL
VAR_INPUT
	// Message location data
	nId			: UINT ; // Identification number of object
	nParentId	: UDINT ; // Id of higher level If aplicable (0 = no parent)
	// Configuration
	fPulsesPerUnit	: LREAL	; // Scale factor for output [units/pulse]
	fOffset			: LREAL	; // Offset for output
	bIcfInverted	: BOOL	; // Invert output position = standard false  
END_VAR
// ====== Set init to true =====
	bInitOk	:= TRUE ; 

// ====== Calculate device id =====
	bInitOk :=	ExecIdentifyDevice(nId,nParentId, E_ComponentTypes.Encoder) AND bInitOk;

// ====== Set manual device type ======
	eDevType := E_Devices.Encoder ;	

	
// ===== copy values to function memory ======
	THIS^.fPulsesPerUnit	:= MAX(fPulsesPerUnit,0.01); // Minimum value of 1
	THIS^.fOffset			:= fOffset;
	THIS^.bIcfInverted		:= bIcfInverted;
END_METHOD

END_FUNCTION_BLOCK

// ---- Encoders/FunctionBlocks/FB_EncoderInput.TcPOU
{attribute 'reflection'}
FUNCTION_BLOCK FB_EncoderInput EXTENDS FB_EncoderBase
VAR_INPUT
END_VAR
VAR_OUTPUT
END_VAR
VAR
	iCounterValue 	AT%I*	: UDINT ;
	iDataError		AT%I*	: BOOL  ;	
	iFrameError		AT%I*	: BOOL  ;
	iPowerFailure	AT%I*	: BOOL  ; 
	iSyncError		AT%I*	: BOOL  ;
	
	nScaledValue		: LREAL ; // Only scaled value for internal use
	nValueWithOffset	: LREAL ; // scaled value with added offset
	fOldPos				: LREAL ; // Old position
	
END_VAR

// ====== Check device status ======
	CheckBoxStatus();

// ====== Scale Output value ======
	nScaledValue := UDINT_TO_LREAL(iCounterValue) / fPulsesPerUnit ;

// ====== Invert ======
	IF bIcfInverted THEN 
		nScaledValue := nScaledValue * -1;
	END_IF
	
// ====== Add offset ======= 
	nValueWithOffset := nScaledValue + fOffset ;
	
// ====== Caclulate velocity =====
	IF Sys_Variables.Pulse100ms THEN 
		nVelocity 	:= (nOutPosition - fOldPos) * 10 ;
		fOldPos		:= nOutPosition;
	END_IF
	
// ====== Set Outputs =======
	nOutPosition 	:= nValueWithOffset ;
	nOutRaw			:= iCounterValue	;

METHOD PRIVATE CheckBoxStatus : BOOL
VAR_INPUT
END_VAR
IF iDataError THEN 
	stFault.Active 			:= TRUE ;
	stFault.Description		:= 'Encoder Data error';
	stFault.FaultType		:= E_FaultTypes.FF;
ELSIF iFrameError THEN 
	stFault.Active 			:= TRUE ;
	stFault.Description		:= 'Encoder frame error';
	stFault.FaultType		:= E_FaultTypes.FF;
ELSIF iPowerFailure THEN 
	stFault.Active 			:= TRUE ;
	stFault.Description		:= 'Encoder Power failure';
	stFault.FaultType		:= E_FaultTypes.FF;
ELSIF iSyncError THEN 
	stFault.Active 			:= TRUE ;
	stFault.Description		:= 'Encoder synchronisation error';
	stFault.FaultType		:= E_FaultTypes.FF;
END_IF
END_METHOD

METHOD PUBLIC FastTask : BOOL
VAR_INPUT
END_VAR
END_METHOD

END_FUNCTION_BLOCK

// ---- Heaters/FB_DevDoublePWM.TcPOU
{attribute 'reflection'}
FUNCTION_BLOCK PUBLIC FB_DevDoublePWM EXTENDS FB_DevBase // PWM control for 2 outputs that cannot be switchid on simultaniously
VAR_INPUT
	bCmdPWMOn			: BOOL := FALSE ; // PWM controller on 
END_VAR
VAR_OUTPUT
END_VAR
VAR
	bCmdChanelAOn		: BOOL := FALSE ; // command switch chanel A on permanently
	bCmdChanelBOn		: BOOL := FALSE ; // Commandswitch chanel B on permanently 
	bCmdOverrulePWM		: BOOL := FALSE ; // Command to overrule PWM
	bCmdHold			: BOOL := false ; // Command hold PWM on signals (collision avoidance)

	tPeriodLength		: TIME  ; // desired PWM cycle time length [ms] 
	tDutyCycle 			: TIME	; // percentage of power [%]
	tIdleTime			: TIME	; // Time both outputs are idle during PWM
	
	tonOutputA 			: TON ; // Timer on PWM output A
	tonOutputB 			: TON ; // Timer on PWM output B
	tonIdle				: TON ; // Timer On PWM Idle time (both outputs off)

	tofOutputA 			: TOF ; // Timer off PWM output A Off (For overlap prevention)
	tofOutputB 			: TOF ; // Timer off PWM output B Off ( for overlap prevention)

	stParPeriodLength	: Udt_Parameter := (fValue := 2000); // desired PWM cycle time length [ms] Parameter
	stParDutyCycle 		: Udt_Parameter	:= ( fValue := 0); // percentage of power [%] Parameter
	stParSwitchOverTime	: Udt_Parameter	; // Time between switching A off and B on (and vice versa) Parameter
	stMaxTimeOn			: Udt_Parameter := (fValue := 1000);// Maximum time a heater can be on without burning through
	
	qbOutputMain AT %Q* 	: BOOL 	; // physical output to main relais
	qbOutputA	 AT %Q* 	: BOOL 	; // physical output to output A
	qbOutputB	 AT %Q* 	: BOOL 	; // physical output to output B
	
	nPWMStep	: INT ; // PWM stepper

	tonBurnTimeA	: TON ; // burn timer for coil A
	tonBurnTimeB	: TON ; // burn timer for coil B 
END_VAR

// set device type
IF eDevType = E_Devices.Undefined THEN 
	eDevType := E_Devices.DoublePWMController ;
END_IF

// Call base function
SUPER^();


// ===== hold all actions if not initialized ======
IF NOT bInitOk THEN
	RETURN;
END_IF 

// call Functions 
CalcCycleTimes();
IF tDutyCycle > T#0S AND tPeriodLength > T#0S THEN // switch PWM controller up when cycle timer is null
	ExecPWMCycle(); // 
END_IF 

ExecSetOutputs();

METHOD INTERNAL CalcCycleTimes : BOOL // calculate cycle timers
VAR_INPUT
END_VAR
VAR 
END_VAR
// Calculate Cycle timers
tPeriodLength	:= LREAL_TO_TIME( stParPeriodLength.fValue );
tDutyCycle		:= LREAL_TO_TIME(stParPeriodLength.fValue * (stParDutyCycle.fValue / 100));
tIdleTime		:= LREAL_TO_TIME(stParPeriodLength.fValue) - (tDutyCycle * 2) ;

tofOutputA.PT := LREAL_TO_TIME(stParSwitchOverTime.fValue);
tofOutputB.PT := LREAL_TO_TIME(stParSwitchOverTime.fValue);
END_METHOD

METHOD PUBLIC CmdHold : BOOL
VAR_INPUT
END_VAR
bCmdHold := TRUE ;

CmdHold := NOT qbOutputMain ;
END_METHOD

METHOD PUBLIC CmdOutputAOn : BOOL // Turn on chanel A permanently 
VAR_INPUT
END_VAR
bCmdOverrulePWM S= TRUE ;
bCmdChanelAOn S= TRUE ;

CmdOutputAOn := qbOutputA AND qbOutputMain ;
END_METHOD

METHOD PUBLIC CmdOutputBOn : BOOL
VAR_INPUT
END_VAR
bCmdOverrulePWM S= TRUE ;
bCmdChanelBOn S= TRUE ;

CmdOutputBOn := qbOutputB AND qbOutputMain ;
END_METHOD

METHOD PUBLIC CmdSafeStop : BOOL
VAR_INPUT
END_VAR
bCmdOverrulePWM S= TRUE ;
bCmdChanelAOn 		:= FALSE ;
bCmdChanelBOn		:= FALSE ;
qbOutputMain 		:= FALSE ;

bIsSafe := NOT (qbOutputA OR qbOutputB OR qbOutputMain);
END_METHOD

METHOD INTERNAL ExecPWMCycle : BOOL
VAR_INPUT
END_VAR
IF bCmdPWMOn THEN 
	IF bCmdOverrulePWM OR bCmdHold THEN 
		IF bCmdChanelAOn THEN 
			nPWMStep := 1 ;
		ELSE 
			nPWMStep := 0 ;
		END_IF
		bCmdOverrulePWM := FALSE ;
		RETURN;
	END_IF
ELSE 
	RETURN;
END_IF

// PWM stepper 
CASE nPWMStep OF 
	0: // Switch on chanel A
		bCmdChanelAOn := TRUE ;
		IF tonOutputA.Q THEN
			nPWMStep := 1 ;
		END_IF
	1: // Switch on chanel B
		bCmdChanelBOn := TRUE;
		IF tonOutputB.Q THEN
			nPWMStep := 2 ;
		END_IF
	2: // Idle Time 
		IF tonIdle.Q THEN 
			nPWMStep := 0;
		END_IF
	ELSE
		;
END_CASE

// call timers 
tonOutputA	(IN := bCmdChanelAOn, PT := tDutyCycle);
tonOutputB	(IN := bCmdChanelBOn, PT := tDutyCycle);
tonIdle 	(IN := nPWMStep = 2	, PT := tIdleTime);
END_METHOD

METHOD PRIVATE ExecSetOutputs : BOOL
VAR_INPUT
END_VAR

// Set main output
qbOutputMain := (bEnable OR bManual) AND NOT bCmdHold ;

// Set outputs
qbOutputA := bCmdChanelAOn AND NOT tofOutputB.Q AND NOT tonBurnTimeA.Q;
qbOutputB := bCmdChanelBOn AND NOT tofOutputA.Q AND NOT tonBurnTimeB.Q;

// Call timers for overlap prevention
tofOutputA(IN := qbOutputA);
tofOutputB(IN := qbOutputB);

// reset commands
bCmdChanelAOn := FALSE ;
bCmdChanelBOn := FALSE ;

tonBurnTimeA ( IN := bCmdChanelAOn, PT := LREAL_TO_TIME( stMaxTimeOn.fValue));
tonBurnTimeB ( IN := bCmdChanelBOn, PT := LREAL_TO_TIME( stMaxTimeOn.fValue));

IF tonBurnTimeA.Q THEN 
	stFault.Active 			:= TRUE ;
	stFault.Description 	:= 'Heater A burn timeout';
	stFault.FaultType		:= E_FaultTypes.CF;
	qbOutputA 				:= FALSE ;
ELSIF tonBurnTimeB.Q THEN 
	stFault.Active 			:= TRUE ;
	stFault.Description 	:= 'Heater B burn timeout';
	stFault.FaultType		:= E_FaultTypes.CF;
	qbOutputB 				:= FALSE ;
END_IF

bCmdHold := FALSE ;
END_METHOD

METHOD PUBLIC Init : BOOL
VAR_INPUT
	// Message location data
	nId			: UINT ; // Identification number of object
	nParentId	: UDINT ; // Id of higher level If aplicable (0 = no parent)
END_VAR
// ====== Set init to true =====
	bInitOk	:= TRUE ; 

// ====== Calculate device id =====
	bInitOk :=	ExecIdentifyDevice(nId,nParentId, E_ComponentTypes.Heaters) AND bInitOk;

// ======= Reset Error bit ======
	bErrorActive 	:= FALSE;
	bBusy			:= FALSE;
	
// ===== configure parameters =====
	stParPeriodLength.fMinimum 		:= 0 		;
	stParPeriodLength.fMaximum		:= 60000 	;
	stParPeriodLength.nNumber 		:= stIdentity.nLocationId + 1;
	stParPeriodLength.sDiscription  := CONCAT( STR1 := stIdentity.sName, STR2 := ' period length of the cycle');
	stParPeriodLength.sName			:= CONCAT( STR1 := stIdentity.sName, STR2 := ' Period Length');
	stParPeriodLength.sType			:= 'MPar';
	stParPeriodLength.sUnit			:= 'ms';
	stParPeriodLength.fValue		:= 5000;

	stParDutyCycle.fMinimum 		:= 0 		;
	stParDutyCycle.fMaximum			:= 50 		;
	stParDutyCycle.nNumber 			:= stIdentity.nLocationId + 2;
	stParDutyCycle.sDiscription  	:= CONCAT( STR1 := stIdentity.sName, STR2 := ' percentage of period length in which an output is active');
	stParDutyCycle.sName			:= CONCAT( STR1 := stIdentity.sName, STR2 := ' Duty Cyle');
	stParDutyCycle.sType			:= 'MPar';
	stParDutyCycle.sUnit			:= '%';
	stParPeriodLength.fValue		:= 10;

	
	stParSwitchOverTime.fMinimum 	:= 0 		;
	stParSwitchOverTime.fMaximum	:= 500 		;
	stParSwitchOverTime.nNumber 	:= stIdentity.nLocationId + 3;
	stParSwitchOverTime.sDiscription:= CONCAT( STR1 := stIdentity.sName, STR2 := ' idle time between output chanel switchover');
	stParSwitchOverTime.sName		:= CONCAT( STR1 := stIdentity.sName, STR2 := ' Switch Time');
	stParSwitchOverTime.sType		:= 'CPar';
	stParSwitchOverTime.sUnit		:= 'ms';

	stMaxTimeOn.fMinimum 	:= 0 		;
	stMaxTimeOn.fMaximum	:= 5000 	;
	stMaxTimeOn.nNumber 	:= stIdentity.nLocationId + 4;
	stMaxTimeOn.sDiscription:= CONCAT( STR1 := stIdentity.sName, STR2 := ' maximum time a heater can be fully on without burning through');
	stMaxTimeOn.sName		:= CONCAT( STR1 := stIdentity.sName, STR2 := ' Max heating time');
	stMaxTimeOn.sType		:= 'MPar';
	stMaxTimeOn.sUnit		:= 'ms';
	
	
	// add parameters to handler 
	refFbParHandler.CmdAddParameter( refParameter := stParPeriodLength );
	refFbParHandler.CmdAddParameter( refParameter := stParDutyCycle );
	refFbParHandler.CmdAddParameter( refParameter := stParSwitchOverTime );
END_METHOD

END_FUNCTION_BLOCK

// ---- Heaters/FB_DevPWMGenerator.TcPOU
{attribute 'reflection'}
FUNCTION_BLOCK PUBLIC FB_DevPWMGenerator EXTENDS FB_DevBase
VAR_INPUT
	nPeriodLength	: DINT	:= 2000 ; // desired PWM cycle time length [ms] 
	nDutyCycle 		: DINT	:= 50 ; // percentage of power [%]
END_VAR
VAR_OUTPUT
END_VAR
VAR
	qbOutput	AT %Q* 	: BOOL 	; // physical output
	bCycleOutput		: BOOL 	; // Cycle output
	tonTimerOn  		: TON 	; // Timer for cycle on
	tofTimerOff			: TOF 	; // timer for cycle off 
	// output commands
	bCmdPWMCycle		: BOOL 	; // run PWM cycle 
	bCmdOn				: BOOL 	; // turn output on permanantly
END_VAR

// Set device type
eDevType := E_Devices.PWMController ;
SUPER^(); 

// calculate cycle times 
CalcCycle();
// set outputs
ExecSetOutput(); 

// reset manual enable
bCmdManual := FALSE ;

METHOD PRIVATE CalcCycle : BOOL
VAR_INPUT
END_VAR
// check if dutycycle is within limits
nDutyCycle := LIMIT(1,nDutyCycle,100);

// Calculate time on from cycle time
tonTimerOn.PT 	:= DINT_TO_TIME(( nPeriodLength / 100) * nDutyCycle);
tofTimerOff.PT	:= DINT_TO_TIME(( nPeriodLength / 100) * (100 - nDutyCycle));
END_METHOD

METHOD PUBLIC CmdOutputCycle : BOOL // start PWM cycle stays on until off command is given
VAR_INPUT
END_VAR
bCmdPWMCycle 	S= TRUE ;
CmdOutputCycle 	:= bCmdPWMCycle ;
END_METHOD

METHOD PUBLIC CmdOutputOff : BOOL // turn off output signal completely
VAR_INPUT
END_VAR
bCmdPWMCycle 	:= FALSE ;
bCmdOn			:= FALSE ;
CmdOutputOff	:= TRUE 	;
END_METHOD

METHOD PUBLIC CmdOutputOn : BOOL // Output stays on until command ends (returns to PWM if active otherwise turns off)
VAR_INPUT
END_VAR
bCmdOn 		S= TRUE ;
CmdOutputOn	:= TRUE ;
END_METHOD

METHOD PRIVATE ExecSetOutput : BOOL
VAR_INPUT
END_VAR

// PWM signal generator
IF bCmdPWMCycle THEN 
	// Run cycle timers 
	tofTimerOff	(IN := tonTimerOn.Q);
	tonTimerOn	(IN := bCycleOutput AND NOT tofTimerOff.Q );
	bCycleOutput := NOT tofTimerOff.Q ;
ELSE
	bCycleOutput := FALSE ;
END_IF

// set output 
IF (bEnable OR bCmdManual) THEN 
	qbOutput := bCycleOutput OR bCmdOn ;
ELSE
	qbOutput := FALSE ;
	RETURN; 
END_IF

// reset continuous on command
bCmdOn := false ;
END_METHOD

METHOD PUBLIC Init : BOOL
VAR_INPUT
	// Location data for messages  
	nId			: UINT ; // Identification number of object
	nParentId	: UDINT ; // Id of higher level If aplicable (0 = no parent)
END_VAR
// ====== Set init to true =====
	bInitOk	:= TRUE ; 

// ====== Calculate device id =====
	bInitOk :=	ExecIdentifyDevice(nId,nParentId, E_ComponentTypes.Heaters) AND bInitOk;
END_METHOD

END_FUNCTION_BLOCK

// ---- Sensors/AnalogInput/FunctionBlocks/FB_DevAnalogInput.TcPOU
{attribute 'reflection'}
FUNCTION_BLOCK PUBLIC FB_DevAnalogInput EXTENDS FB_DevBase
VAR_INPUT
	bCmdSimulate	: BOOL 	:= FALSE ;// Simulate sensor Input 
	fSimValue		: INT	:= 0 ;// Simulated sensor state
END_VAR
VAR_OUTPUT
	fValue	: LREAL := 0 ; // Input value from hardware (converted to LREAL)
END_VAR
VAR
	inHwInput 	AT%I* : INT ; // Hardware connection
	inStatus	AT%I* : BYTE; // input card hardware status
END_VAR

// Set device type
eDevType := E_Devices.AnalogSensor ;

// Call base function
SUPER^();

// Check Hardware connection
CheckHardware();
// set feedback
ExecSetFeedback();

// Make sure compiler does not skip unused variables

METHOD CheckHardware : BOOL
VAR_INPUT
END_VAR
// Check for hardware faults
IF inStatus.0 THEN // signal under range
	stFault.Active			:= TRUE 							;
	stFault.Description		:= 'Signal under range';
	stFault.FaultType		:= E_FaultTypes.CF 					;
	bErrorActive			:= TRUE 							;
END_IF

IF inStatus.1 THEN // signal over range
	stFault.Active			:= TRUE 							;
	stFault.Description		:= 'Signal over range';
	stFault.FaultType		:= E_FaultTypes.CF 					;
	bErrorActive			:= TRUE 							;
END_IF

IF inStatus.6 THEN // general error bit
	stFault.Active			:= TRUE 							;
	stFault.Description		:= 'Hardware General Error';
	stFault.FaultType		:= E_FaultTypes.FF 					;
	bErrorActive			:= TRUE 							;
END_IF
END_METHOD

METHOD ExecSetFeedback : BOOL
VAR_INPUT
END_VAR
IF bCmdSimulate THEN 
	fValue := int_to_lreal(fSimValue) ;
ELSE
	fValue := INT_TO_LREAL(inHwInput);
END_IF

ExecSetFeedback := TRUE;
END_METHOD

METHOD PUBLIC Init : BOOL
VAR_INPUT
	// Location data for messages  
	nId			: UINT ; // Identification number of object
	nParentId	: UDINT ; // Id of higher level If aplicable (0 = no parent)
END_VAR
// ====== Set init to true =====
	bInitOk	:= TRUE ; 

// ====== Calculate device id =====
	bInitOk :=	ExecIdentifyDevice(nId,nParentId, E_ComponentTypes.AnInput) AND bInitOk;

// ====== Set feedback =====
	Init := bInitOk ;
END_METHOD

END_FUNCTION_BLOCK

// ---- Sensors/AnalogInput/FunctionBlocks/FB_DevAnalogInputScaled.TcPOU
{attribute 'reflection'}
FUNCTION_BLOCK PUBLIC FB_DevAnalogInputScaled EXTENDS FB_DevAnalogInput
VAR_INPUT
END_VAR
VAR_OUTPUT
END_VAR
VAR
	nLimitMin		: INT := IBF_Utilities.GVL_FixedValues.nINTMINVALUE	; // Initial value is set to integer minimum value for use with normal def analog inputs 
	nLimitMax 		: INT := IBF_Utilities.GVL_FixedValues.nINTMAXVALUE	; // Initial value is set to integer minimum value for use with high def analog inputs
	fGainFactor 	: LREAL	:= 1	;
	nOfset			: INT	:= 0	;
END_VAR

SUPER^();

METHOD ExecSetFeedback : BOOL
VAR
	nCalibValue	: INT ; 
END_VAR
// Offset 
IF bCmdSimulate THEN 
	nCalibValue := fSimValue + nOfset ;
ELSE
	nCalibValue := inHwInput + nOfset ;
END_IF

fValue := INT_TO_LREAL(nCalibValue) / fGainFactor;

ExecSetFeedback := TRUE;
END_METHOD

METHOD PUBLIC SetScaling : BOOL 
VAR_INPUT
	fMaxValue	: LREAL ; 	// Maximum input value after scaling, e.g. 100%, 0 = no scaling (gain = hardware limit / fMaxValue)  
	fOfset		: LREAL ;	// offset value (fvalue = (gain * hwvalue) + fOfset)
END_VAR
// calculate gain 
IF fMaxValue =0 THEN 
	fGainFactor := 1 ;
ELSE 
	fGainFactor := nLimitMax / fMaxValue ;
END_IF

nOfset := LREAL_TO_INT(fOfset * fGainFactor) ;

SetScaling := TRUE;
END_METHOD

END_FUNCTION_BLOCK

// ---- Sensors/AnalogInput/FunctionBlocks/FB_DevHDAnalogInAutoCalibrate.TcPOU
{attribute 'reflection'}
FUNCTION_BLOCK PUBLIC FB_DevHDAnalogInAutoCalibrate EXTENDS FB_DevHDAnalogInputScaled
VAR_INPUT
END_VAR
VAR_OUTPUT
END_VAR
VAR
END_VAR

SUPER^();

METHOD PUBLIC CmdCalibrateNull : BOOL
VAR_INPUT
END_VAR
// set offset to calibrate to null
nOfset := - inHwInput ;

CmdCalibrateNull := TRUE;
END_METHOD

METHOD PUBLIC CmdCalilbrateValue : BOOL // calibrate gain factor to actual value (warning calibrate to null before calibrating to value)
VAR_INPUT
	fCalibrationValue	: LREAL ; // Active input value to sensor (calibration setpoint)
END_VAR
// set gain from current value
fGainFactor := DINT_TO_LREAL(inHwInput + nOfset) / fCalibrationValue ; 

CmdCalilbrateValue := TRUE;
END_METHOD

END_FUNCTION_BLOCK

// ---- Sensors/AnalogInput/FunctionBlocks/FB_DevHDAnalogInputScaled.TcPOU
{attribute 'reflection'}
FUNCTION_BLOCK PUBLIC FB_DevHDAnalogInputScaled EXTENDS FB_DevHDAnalogInput
VAR_INPUT
END_VAR
VAR_OUTPUT
END_VAR
VAR
	fGainFactor 	: LREAL	:= 1	;
	nOfset			: DINT	:= 0	;
END_VAR

SUPER^();

METHOD ExecSetFeedback : BOOL
VAR
	nCalibValue	: DINT ; 
END_VAR
// Offset 
IF bCmdSimulate THEN 
	nCalibValue := fSimValue + nOfset ;
ELSE
	nCalibValue := inHwInput + nOfset ;
END_IF

fValue := DINT_TO_LREAL(nCalibValue) / fGainFactor;

ExecSetFeedback := TRUE;
END_METHOD

METHOD PUBLIC SetScaling : BOOL 
VAR_INPUT
	fMaxValue	: LREAL ; 	// Maximum input value after scaling, e.g. 100%, 0 = no scaling (gain = hardware limit / fMaxValue)  
	fOfset		: LREAL ;	// offset value (fvalue = (gain * hwvalue) + fOfset)
END_VAR
// calculate gain 
IF fMaxValue =0 THEN 
	fGainFactor := 1 ;
ELSE 
	fGainFactor := nLimitMax / fMaxValue ;
END_IF

nOfset := LREAL_TO_DINT(fOfset * fGainFactor) ;

SetScaling := TRUE;
END_METHOD

END_FUNCTION_BLOCK

// ---- Sensors/AnalogInput/FunctionBlocks/FB_DevHDAnalogInput.TcPOU
{attribute 'reflection'}
FUNCTION_BLOCK PUBLIC FB_DevHDAnalogInput EXTENDS FB_DevBase
VAR_INPUT
	bCmdSimulate	: BOOL 	:= FALSE ;// Simulate sensor Input 
	fSimValue		: DINT	:= 0 ;// Simulated sensor state
END_VAR
VAR_OUTPUT
	fValue	: LREAL := 0 ; // Analog input value (LREAL)
END_VAR
VAR
	nLimitMin			: DINT := IBF_Utilities.GVL_FixedValues.nDINTMINVALUE	; // Initial value is set to integer minimum value for use with normal def analog inputs 
	nLimitMax 			: DINT := IBF_Utilities.GVL_FixedValues.nDINTMAXVALUE 	; // Initial value is set to integer minimum value for use with high def analog inputs
	inHwInput 	AT%I* 	: DINT ; // Hardware connection
	inStatus	AT%I* 	: BYTE; // input card hardware status
END_VAR

// Set device type
eDevType := E_Devices.AnalogSensor ;

// Call base function
SUPER^();

// Check Hardware connection
CheckHardware();

// set feedback
ExecSetFeedback();

METHOD CheckHardware : BOOL
VAR_INPUT
END_VAR
// Check for hardware faults
IF inStatus.0 THEN // signal under range
	stFault.Active			:= TRUE 							;
	stFault.Description		:= 'Signal under Range';
	stFault.FaultType		:= E_FaultTypes.CF 					;
	bErrorActive			:= TRUE 							;
END_IF

IF inStatus.1 THEN // signal over range
	stFault.Active			:= TRUE 							;
	stFault.Description		:= 'Signal over Range';
	stFault.FaultType		:= E_FaultTypes.CF 					;
	bErrorActive			:= TRUE 							;
END_IF

IF inStatus.6 THEN // general Error bit
	stFault.Active			:= TRUE 							;
	stFault.Description		:= 'Hardware general Error';
	stFault.FaultType		:= E_FaultTypes.FF 					;
	bErrorActive			:= TRUE 							;
END_IF
END_METHOD

METHOD ExecSetFeedback : BOOL
VAR_INPUT
END_VAR
IF bCmdSimulate THEN 
	fValue := fSimValue ;
ELSE
	fValue := DINT_TO_LREAL(inHwInput);
END_IF

ExecSetFeedback := TRUE;
END_METHOD

METHOD PUBLIC Init : BOOL
VAR_INPUT
	// Location data for messages  
	nId			: UINT ; // Identification number of object
	nParentId	: UDINT ; // Id of higher level If aplicable (0 = no parent)
END_VAR
// ====== Set init to true =====
	bInitOk	:= TRUE ; 

// ====== Calculate device id =====
	bInitOk :=	ExecIdentifyDevice(nId,nParentId, E_ComponentTypes.AnInput) AND bInitOk;

// ====== Set feedback =====
	Init := bInitOk ;
END_METHOD

END_FUNCTION_BLOCK

// ---- Sensors/AnalogInput/FunctionBlocks/FB_DevAnalogInAutoCalibrate.TcPOU
{attribute 'reflection'}
FUNCTION_BLOCK PUBLIC FB_DevAnalogInAutoCalibrate EXTENDS FB_DevAnalogInputScaled
VAR_INPUT
END_VAR
VAR_OUTPUT
END_VAR
VAR
END_VAR

SUPER^();

METHOD PUBLIC CmdCalibrateNull : BOOL
VAR_INPUT
END_VAR
// set offset to calibrate to null
nOfset := - inHwInput ;

CmdCalibrateNull := TRUE;
END_METHOD

METHOD PUBLIC CmdCalilbrateValue : BOOL // calibrate gain factor to actual value (warning calibrate to null before calibrating to value)
VAR_INPUT
	fCalibrationValue	: LREAL ; // Active input value to sensor (calibration setpoint)
END_VAR
// set gain from current value
fGainFactor := INT_TO_LREAL(inHwInput + nOfset) / fCalibrationValue ; 

CmdCalilbrateValue := TRUE;
END_METHOD

END_FUNCTION_BLOCK

// ---- Sensors/FootPedals/FunctionBlocks/FB_EfkaEB301A_FootPedal.TcPOU
{attribute 'reflection'}
FUNCTION_BLOCK PUBLIC FB_EfkaEB301A_FootPedal EXTENDS FB_DevBase
VAR_OUTPUT
	ePedalInputStep		: E_FootpedalPos	:= 0 ;
	bRTrigtoReverse1 	: BOOL := FALSE ; // rising edge trigger when pedal moves from 0 to -1 or Idle to reverse 1 
	bRTrigtoReverse2 	: BOOL := FALSE ; // rising edge trigger when pedal moves from 1 to -2 or reverse 1 to reverse 2 
	bRTrigtoForward1 	: BOOL := FALSE ; // rising edge trigger when pedal moves from 0 to 1 or idle to forward 1 
	bRTrigtoForward2 	: BOOL := FALSE ; // rising edge trigger when pedal moves from 0 to 1 or forward to forward 2 
END_VAR
VAR
	// ===== greycode switches from footpedal =====
	I_GreyCodeA AT%I* : BOOL	; // Greycode input a from foot pedal 
	I_GreyCodeB AT%I* : BOOL	; // Greycode input a from foot pedal 
	I_GreyCodeC AT%I* : BOOL	; // Greycode input a from foot pedal 
	I_GreyCodeD AT%I* : BOOL	; // Greycode input a from foot pedal 
	nGreyCodetotal	: BYTE ; // all greycode switches combined
	// ==== decimal value =====
	ePreviousPedalInput	: E_FootpedalPos	:= 0 ;
END_VAR

// ===== Read input from pedal =====
ACT_ConvertGreycode();

// ===== Create edge flanks for functions =====
ACT_CreateEdges();

ACTION ACT_ConvertGreycode:
// ===== Combine greycode sensors =====
nGreyCodetotal.0 := I_GreyCodeA ;
nGreyCodetotal.1 := I_GreyCodeB ;
nGreyCodetotal.2 := I_GreyCodeC ;
nGreyCodetotal.3 := I_GreyCodeD ;

// ==== Convert greycode decimal to speed steps =====
// this only makes sense in EFKA world but anyway let's convert it to our own sense

CASE nGreyCodetotal OF 								  // DCBA
	03: ePedalInputStep := E_FootpedalPos.eReverse2	; // 0011
	01: ePedalInputStep := E_FootpedalPos.eReverse1	; // 0001
	00: ePedalInputStep := E_FootpedalPos.eIdle		; // 0000
	02: ePedalInputStep := E_FootpedalPos.eForward0	; // 0010
	06: ePedalInputStep := E_FootpedalPos.eForward1	; // 0110
 	07: ePedalInputStep := E_FootpedalPos.eForward2	; // 0111
	05: ePedalInputStep := E_FootpedalPos.eForward3	; // 0101
	04: ePedalInputStep := E_FootpedalPos.eForward4	; // 0100
	12:	ePedalInputStep := E_FootpedalPos.eForward5	; // 1100
	13:	ePedalInputStep := E_FootpedalPos.eForward6	; // 1101
	15: ePedalInputStep := E_FootpedalPos.eForward7	; // 1111
	14: ePedalInputStep := E_FootpedalPos.eForward8	; // 1110
	10: ePedalInputStep := E_FootpedalPos.eForward9	; // 1010
	11: ePedalInputStep := E_FootpedalPos.eForward10; // 1011
	09: ePedalInputStep := E_FootpedalPos.eForward11; // 1001
	08: ePedalInputStep := E_FootpedalPos.eForward12; // 1000
	ELSE
		ePedalInputStep := E_FootpedalPos.eFalse 	;
END_CASE
END_ACTION

ACTION ACT_CreateEdges:
// ===== create edges on which functions can be triggerd =====
CASE ePedalInputStep OF
	E_FootpedalPos.eReverse2:
		bRTrigtoReverse2 := ePreviousPedalInput = E_FootpedalPos.eReverse1 ;
	E_FootpedalPos.eReverse1:
		bRTrigtoReverse1 := ePreviousPedalInput = E_FootpedalPos.eIdle ;
	E_FootpedalPos.eForward0:
		bRTrigtoForward1 := ePreviousPedalInput = E_FootpedalPos.eIdle ;
	E_FootpedalPos.eForward1: 
		bRTrigtoForward2 := ePreviousPedalInput = E_FootpedalPos.eForward0 ; 
END_CASE 

// write previous pedal input 
ePreviousPedalInput := ePedalInputStep ;
END_ACTION

METHOD PUBLIC Init : BOOL
VAR_INPUT
	// Location data for messages  
	nId			: UINT ; // Identification number of object
	nParentId	: UDINT ; // Id of higher level If aplicable (0 = no parent)
END_VAR
// ====== Set init to true =====
	bInitOk	:= TRUE ; 

// ====== Calculate device id =====
	bInitOk :=	ExecIdentifyDevice(nId,nParentId, E_ComponentTypes.NA) AND bInitOk;

// ====== Set feedback =====
	Init := bInitOk;
END_METHOD

END_FUNCTION_BLOCK

// ---- GlobalTextList.TcGTLO
TEXTLIST GlobalTextList
  0 = ' Act velocity:'
  222 = '%f'
  388 = '%i'
  568 = '%n'
  596 = '%s'
  224 = 'Activate manual control'
  584 = 'Actual Position:'
  252 = 'Actual velocity:'
  120 = 'Admin'
  614 = 'CCW'
  447 = 'CCW Fast'
  50 = 'Close'
  825 = 'Command distance:'
  263 = 'Command Position:'
  851 = 'Command velocity:'
  1 = 'component fault active'
  641 = 'CW'
  297 = 'CW Fast'
  626 = 'Cycle Time [ms]'
  1062 = 'Deactivate manual control'
  740 = 'Duty cycle [%]'
  422 = 'Enable manual control'
  274 = 'Home'
  445 = 'Homed:'
  546 = 'Input value: %i'
  879 = 'Jog Forward'
  223 = 'Jog Inching'
  370 = 'Jog reverse'
  7 = 'Light blink fast'
  137 = 'Light blink slow'
  616 = 'Light On'
  145 = 'Login'
  990 = 'Logout'
  804 = 'Manual control active'
  345 = 'ManualControl'
  948 = 'Move to target position'
  356 = 'Moving:'
  33 = 'None'
  313 = 'ON'
  463 = 'Open'
  674 = 'Operator'
  425 = 'Output A'
  527 = 'Output A on'
  808 = 'Output B'
  110 = 'Output B On'
  39 = 'Output value:'
  703 = 'ParameterControl'
  704 = 'Pulse'
  174 = 'Reset'
  559 = 'Run CCW'
  493 = 'Run Clockwise'
  220 = 'Run Clockwise Fast'
  212 = 'Run Counter clockwise'
  691 = 'Run Counter clockwise Fast'
  928 = 'Run CW'
  400 = 'Select device'
  838 = 'Service'
  320 = 'Set Value'
  771 = 'Teach'
  553 = 'Time to close [ms]'
  243 = 'Time to open [ms]'
  344 = 'User mgmt'
END_TEXTLIST

// ---- GroupHandlers/ManualControlHandler/HMI/DeviceScreens/VisuAnalogAxisControl.TcVIS
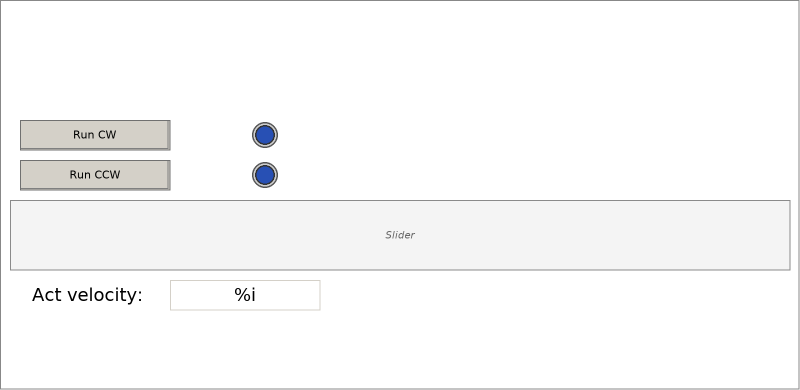
VISUALIZATION VisuAnalogAxisControl  // 800x390
VAR_IN_OUT
	pDev : POINTER TO FB_DevAnalogAxis;
END_VAR
    Slider (10,200 780x70), variable: pDev^.stManualCtrl.fCmdVelocity, scale 0..100
    Textfield (170,280 150x30), "%i", text variable: pDev^.fActVelocity
        OnMouseClick: write the text variable via VisuDialogs.Numpad
    Label (10,280 150x30), "Act velocity:"
    Button (20,120 150x30), "Run CW"
        tap pDev^.stManualCtrl.bCmdRunCW
    Button (20,160 150x30), "Run CCW"
        tap pDev^.stManualCtrl.bCmdRunCCW
    Lamp1 (190,120 150x30), variable: pDev^.bMovingCW, style: Lamp-Lamp1-Blue
    Lamp1 (190,160 150x30), variable: pDev^.bMovingCCW, style: Lamp-Lamp1-Blue
END_VISUALIZATION

// ---- GroupHandlers/ManualControlHandler/HMI/DeviceScreens/VisuAnalogOutControl.TcVIS
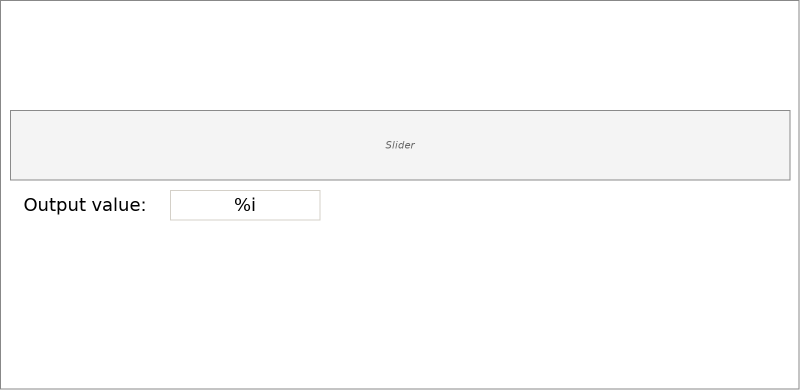
VISUALIZATION VisuAnalogOutControl  // 800x390
VAR_IN_OUT
	pDev : POINTER TO FB_DevAnalogOutput;
END_VAR
    Slider (10,110 780x70), variable: pDev^.fCmdValue, scale 0..100
    Textfield (170,190 150x30), "%i", text variable: pDev^.fCmdValue
        OnMouseClick: write the text variable via VisuDialogs.Numpad
    Label (10,190 150x30), "Output value:"
END_VISUALIZATION

// ---- GroupHandlers/ManualControlHandler/HMI/DeviceScreens/VisuAnlogInputControl.TcVIS
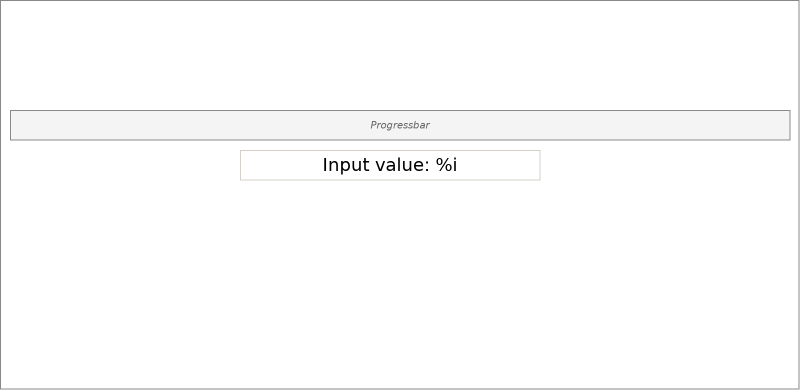
VISUALIZATION VisuAnlogInputControl  // 800x390
VAR_IN_OUT
	pDev : POINTER TO FB_DevAnalogInput;
END_VAR
    Progressbar (10,110 780x30), variable: pDev^.fValue
    Textfield (240,150 300x30), "Input value: %i", text variable: pDev^.fValue
END_VISUALIZATION

// ---- GroupHandlers/ManualControlHandler/HMI/DeviceScreens/VisuAxisControl.TcVIS
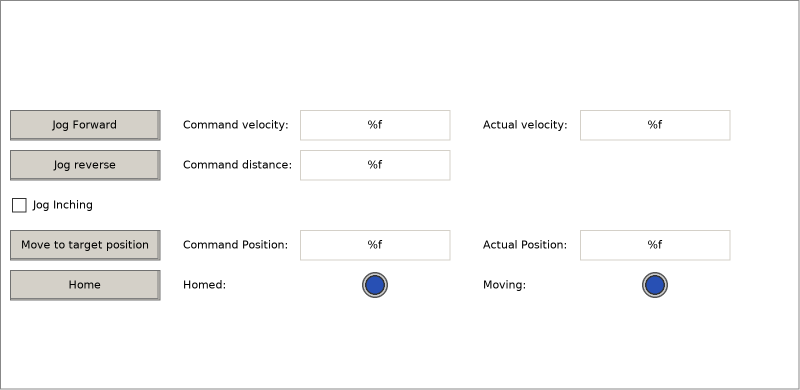
VISUALIZATION VisuAxisControl  // 800x390
VAR_IN_OUT
	pDev : POINTER TO Fb_DevAxis; 
END_VAR
    Button (10,110 150x30), "Jog Forward"
        tap pDev^.stManualCtrl.bCmdJogForward
    Button (10,150 150x30), "Jog reverse"
        tap pDev^.stManualCtrl.bCmdJogReverse
    Button (10,230 150x30), "Move to target position"
        tap pDev^.stManualCtrl.bCmdToPos
    Button (10,270 150x30), "Home"
        tap pDev^.stManualCtrl.bCmdHome
    Checkbox (10,190 150x30), "Jog Inching", variable: pDev^.stManualCtrl.bCmdInching
    Label (180,150 120x30), "Command distance:"
    Label (180,110 120x30), "Command velocity:"
    Label (180,230 120x30), "Command Position:"
    Textfield (300,110 150x30), "%f", text variable: pDev^.stManualCtrl.fVelocity
        OnMouseDown: write the text variable via VisuDialogs.Numpad
    Textfield (300,150 150x30), "%f", text variable: pDev^.stManualCtrl.fDistance
        OnMouseDown: write the text variable via VisuDialogs.Numpad
    Textfield (300,230 150x30), "%f", text variable: pDev^.stManualCtrl.fPosition
        OnMouseDown: write the text variable via VisuDialogs.Numpad
    Label (480,110 100x30), "Actual velocity:"
    Label (480,230 100x30), "Actual Position:"
    Textfield (580,230 150x30), "%f", text variable: pDev^.fActPosition
        OnMouseDown: write the text variable via VisuDialogs.Numpad
    Textfield (580,110 150x30), "%f", text variable: pDev^.fVelocity
        OnMouseDown: write the text variable via VisuDialogs.Numpad
    Lamp1 (580,270 150x30), variable: pDev^.AxisRef.Status.Moving, style: Lamp-Lamp1-Blue
    Label (480,270 100x30), "Moving:"
    Lamp1 (300,270 150x30), variable: pDev^.AxisRef.Status.Homed, style: Lamp-Lamp1-Blue
    Label (180,270 120x30), "Homed:"
END_VISUALIZATION

// ---- GroupHandlers/ManualControlHandler/HMI/DeviceScreens/VisuCylinderControl.TcVIS
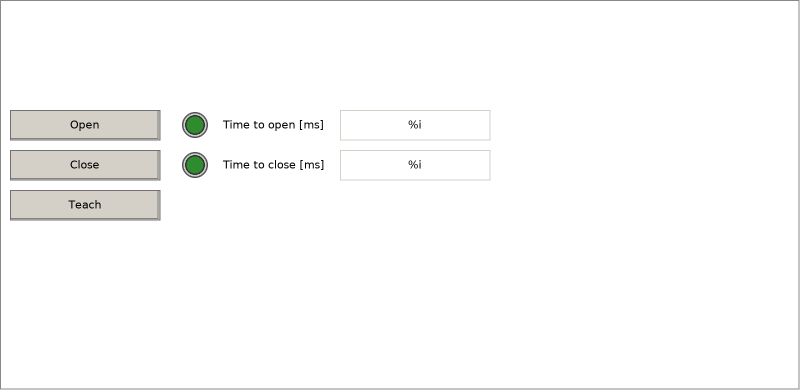
VISUALIZATION VisuCylinderControl  // 800x390
VAR_IN_OUT
	pDev : POINTER TO Fb_DevCylWithFbk; 
END_VAR
    Button (10,110 150x30), "Open"
        tap pDev^.stManualCtrl.bCmdOpen
    Button (10,150 150x30), "Close"
        tap pDev^.stManualCtrl.bCmdClose
    Lamp1 (180,110 30x30), variable: pDev^.bFco_Open, style: Lamp-Lamp1-Green
    Button (10,190 150x30), "Teach"
        toggle pDev^.stManualCtrl.bCmdTeach
    Lamp1 (180,150 30x30), variable: pDev^.bFco_Closed, style: Lamp-Lamp1-Green
    Label (220,110 100x30), "Time to open [ms]"
    Label (220,150 100x30), "Time to close [ms]"
    Textfield (340,150 150x30), "%i", text variable: pDev^.stParTimeToClose.fValue
        OnMouseClick: write the text variable via VisuDialogs.Numpad, min 0
    Textfield (340,110 150x30), "%i", text variable: pDev^.stParTimeToOpen.fValue
        OnMouseClick: write the text variable via VisuDialogs.Numpad, min 0
END_VISUALIZATION

// ---- GroupHandlers/ManualControlHandler/HMI/DeviceScreens/VisuDigitalInputControl.TcVIS
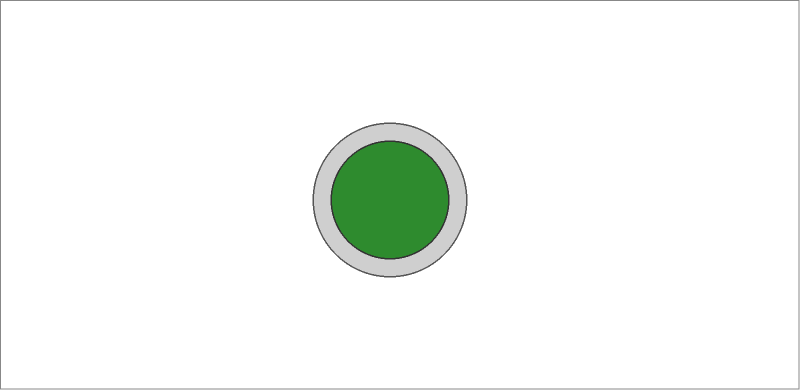
VISUALIZATION VisuDigitalInputControl  // 800x390
VAR_IN_OUT
	pDev : POINTER TO Fb_DevDigitalInputFunctions;
END_VAR
    Lamp1 (300,110 180x180), variable: pDev^.bFcoInputActive, style: Lamp-Lamp1-Green
END_VISUALIZATION

// ---- GroupHandlers/ManualControlHandler/HMI/DeviceScreens/VisuDigitalOutControl.TcVIS
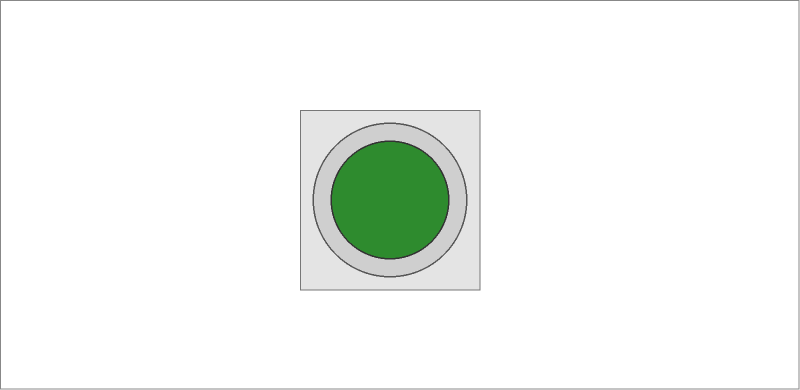
VISUALIZATION VisuDigitalOutControl  // 800x390
VAR_IN_OUT
	pDev : POINTER TO FB_DevDigitalOutput;
END_VAR
    PushSwitch (300,110 180x180), variable: pDev^.bCmdOn, behaviour: TOGGLE, style: Switch-PushSwitch-Green
END_VISUALIZATION

// ---- GroupHandlers/ManualControlHandler/HMI/DeviceScreens/VisuDoublePWMControl.TcVIS
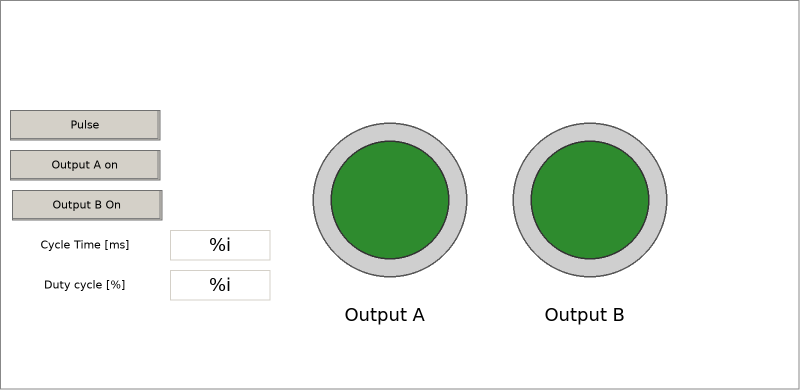
VISUALIZATION VisuDoublePWMControl  // 800x390
VAR_IN_OUT
	pDev : POINTER TO FB_DevDoublePWM;
END_VAR
    Lamp1 (300,110 180x180), variable: pDev^.qbOutputA, style: Lamp-Lamp1-Green
    Button (10,110 150x30), "Pulse"
        toggle pDev^.bCmdPWMOn
    Button (10,150 150x30), "Output A on"
        toggle pDev^.bCmdChanelAOn
    Textfield (170,230 100x30), "%i", text variable: pDev^.stParPeriodLength.fValue
        OnMouseUp: write the text variable via VisuDialogs.Numpad
    Label (10,230 150x30), "Cycle Time [ms]"
    Label (10,270 150x30), "Duty cycle [%]"
    Textfield (170,270 100x30), "%i", text variable: pDev^.stParDutyCycle.fValue
        OnMouseClick: write the text variable via VisuDialogs.Numpad, min 0, max 100
    Lamp1 (500,110 180x180), variable: pDev^.qbOutputB, style: Lamp-Lamp1-Green
    Button (12,190 150x30), "Output B On"
        tap pDev^.bCmdChanelBOn
    Label (310,300 150x30), "Output A"
    Label (510,300 150x30), "Output B"
END_VISUALIZATION

// ---- GroupHandlers/ManualControlHandler/HMI/DeviceScreens/VisuEncoderInput.TcVIS
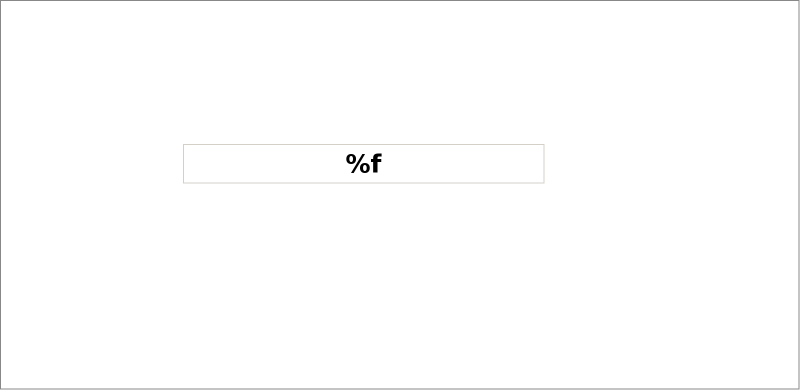
VISUALIZATION VisuEncoderInput  // 800x390
VAR_IN_OUT
	pDev : POINTER TO FB_EncoderBase;
END_VAR
    Textfield (183,144 361x39), "%f", text variable: pDev^.nOutPosition
END_VISUALIZATION

// ---- GroupHandlers/ManualControlHandler/HMI/DeviceScreens/VisuKL15XXControl.TcVIS
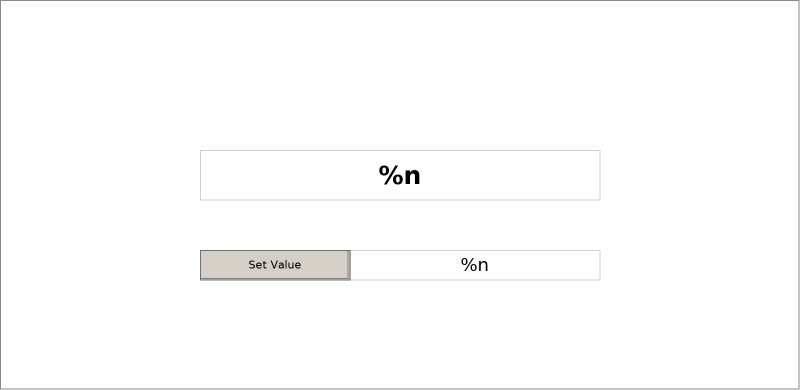
VISUALIZATION VisuKL15XXControl  // 800x390
VAR_IN_OUT
	pDev : POINTER TO FB_DevKL1512;
END_VAR
    Textfield (200,150 400x50), "%n", text variable: pDev^.stManualControl.nCount
    Textfield (350,250 250x30), "%n", text variable: pDev^.stManualControl.nManValue
        OnMouseClick: write the text variable via VisuDialogs.Numpad
    Button (200,250 150x30), "Set Value"
        tap pDev^.stManualControl.bManSetValue
END_VISUALIZATION

// ---- GroupHandlers/ManualControlHandler/HMI/DeviceScreens/VisuKL5151Control.TcVIS
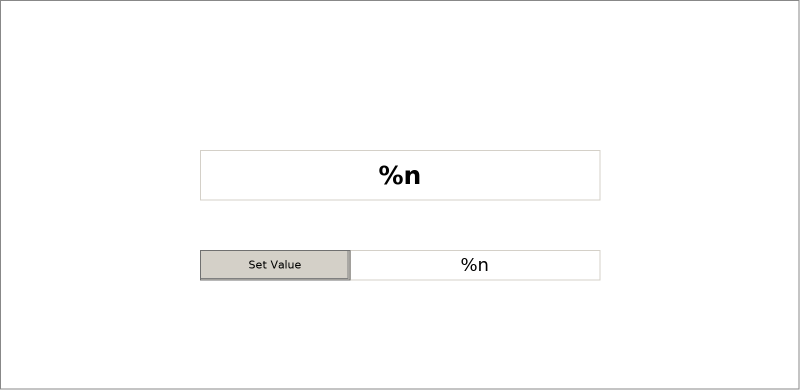
VISUALIZATION VisuKL5151Control  // 800x390
VAR_IN_OUT
	pDev : POINTER TO FB_DevKL5151;
END_VAR
    Textfield (200,150 400x50), "%n", text variable: pDev^.stManualControl.nCount
    Textfield (350,250 250x30), "%n", text variable: pDev^.stManualControl.nManValue
        OnMouseClick: write the text variable via VisuDialogs.Numpad
    Button (200,250 150x30), "Set Value"
        tap pDev^.stManualControl.bManSetValue
END_VISUALIZATION

// ---- GroupHandlers/ManualControlHandler/HMI/DeviceScreens/VisuPushbuttonLightControl.TcVIS
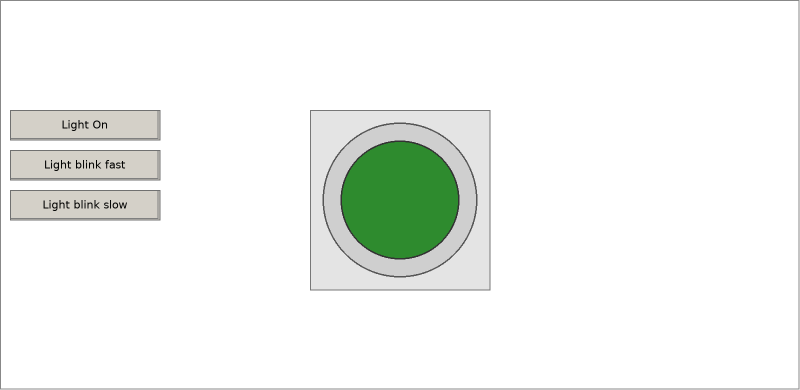
VISUALIZATION VisuPushbuttonLightControl  // 800x390
VAR_IN_OUT
	pDev : POINTER TO FB_DevPushbuttonLight;
END_VAR
    PushSwitch (310,110 180x180), variable: pDev^.bFcoInputActive, behaviour: TOGGLE, style: Switch-PushSwitch-Green
    Button (10,110 150x30), "Light On"
        toggle pDev^.fbLight.bCmdOn
    Button (10,150 150x30), "Light blink fast"
        toggle pDev^.fbLight.bCmdBlinkFast
    Button (10,190 150x30), "Light blink slow"
        toggle pDev^.fbLight.bCmdBlinkSlow
END_VISUALIZATION

// ---- GroupHandlers/ManualControlHandler/HMI/DeviceScreens/VisuPWMControl.TcVIS
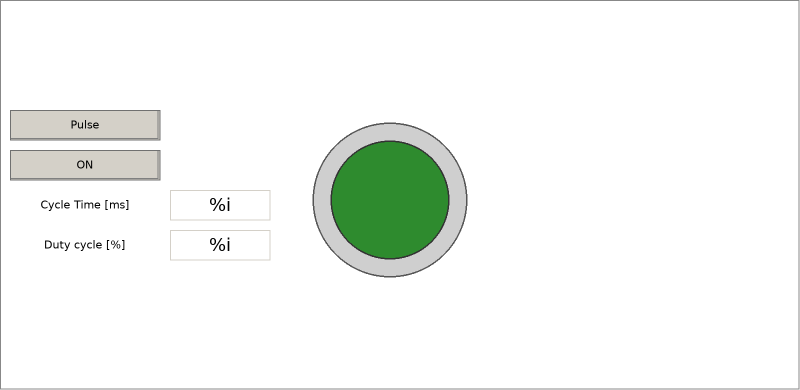
VISUALIZATION VisuPWMControl  // 800x390
VAR_IN_OUT
	pDev : POINTER TO FB_DevPWMGenerator;
END_VAR
    Lamp1 (300,110 180x180), variable: pDev^.qbOutput, style: Lamp-Lamp1-Green
    Button (10,110 150x30), "Pulse"
        toggle pDev^.bCmdPWMCycle
    Button (10,150 150x30), "ON"
        tap pDev^.bCmdOn
    Textfield (170,190 100x30), "%i", text variable: pDev^.nPeriodLength
        OnMouseUp: write the text variable via VisuDialogs.Numpad
    Label (10,190 150x30), "Cycle Time [ms]"
    Label (10,230 150x30), "Duty cycle [%]"
    Textfield (170,230 100x30), "%i", text variable: pDev^.nDutyCycle
        OnMouseClick: write the text variable via VisuDialogs.Numpad, min 0, max 100
END_VISUALIZATION

// ---- GroupHandlers/ManualControlHandler/HMI/DeviceScreens/VisuTwoVelocityAxisControl.TcVIS
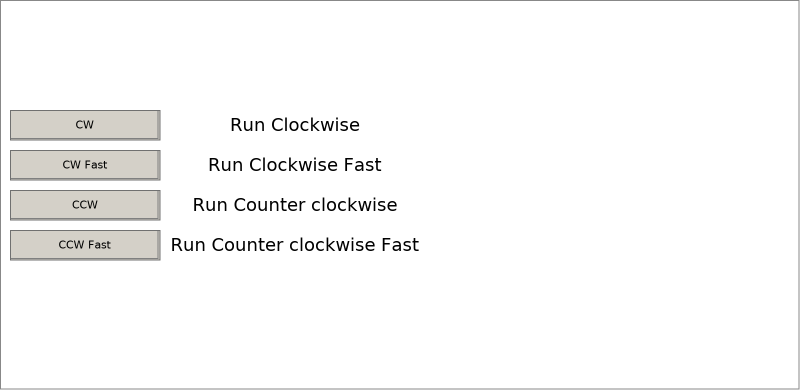
VISUALIZATION VisuTwoVelocityAxisControl  // 800x390
VAR_IN_OUT
	pDev : POINTER TO FB_DevTwoVelocityAxis;
END_VAR
    Button (10,110 150x30), "CW"
        tap pDev^.stManualControl.bManRunCW
    Button (10,150 150x30), "CW Fast"
        tap pDev^.stManualControl.bManRunCWFast
    Button (10,190 150x30), "CCW"
        tap pDev^.stManualControl.bManRunCCw
    Button (10,230 150x30), "CCW Fast"
        tap pDev^.stManualControl.bManRunCCWFast
    Label (170,110 250x30), "Run Clockwise"
    Label (170,150 250x30), "Run Clockwise Fast"
    Label (170,190 250x30), "Run Counter clockwise"
    Label (170,230 250x30), "Run Counter clockwise Fast"
END_VISUALIZATION

// ---- GroupHandlers/ManualControlHandler/HMI/DeviceScreens/VisuUndefinedControl.TcVIS
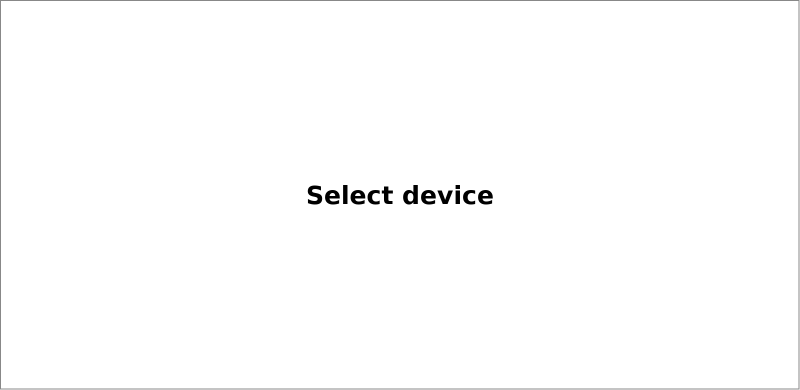
VISUALIZATION VisuUndefinedControl  // 800x390
    Label (0,0 800x390), "Select device"
END_VISUALIZATION

// ---- GroupHandlers/ManualControlHandler/HMI/DeviceScreens/VisuValveControl.TcVIS
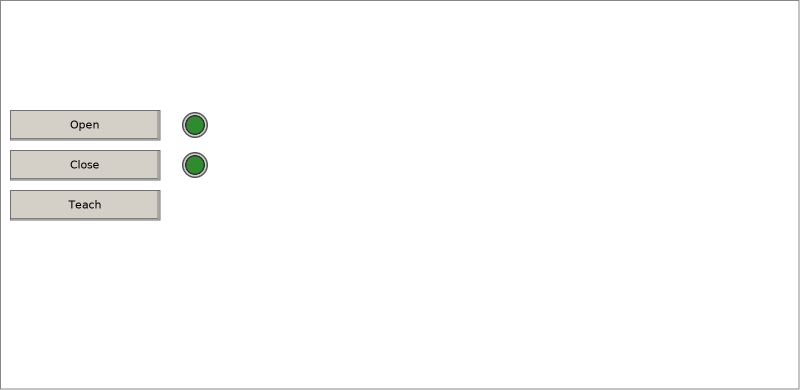
VISUALIZATION VisuValveControl  // 800x390
VAR_IN_OUT
	pDev : POINTER TO FB_DevValve;
END_VAR
    Button (10,110 150x30), "Open"
        tap pDev^.stManualCtrl.bCmdOpen
    Button (10,150 150x30), "Close"
        tap pDev^.stManualCtrl.bCmdClose
    Lamp1 (180,110 30x30), variable: pDev^.bFco_Open, style: Lamp-Lamp1-Green
    Button (10,190 150x30), "Teach"
        toggle pDev^.stManualCtrl.bCmdTeach
    Lamp1 (180,150 30x30), variable: pDev^.bFco_Closed, style: Lamp-Lamp1-Green
END_VISUALIZATION

// ---- GroupHandlers/ManualControlHandler/HMI/ManualControl.TcVIS
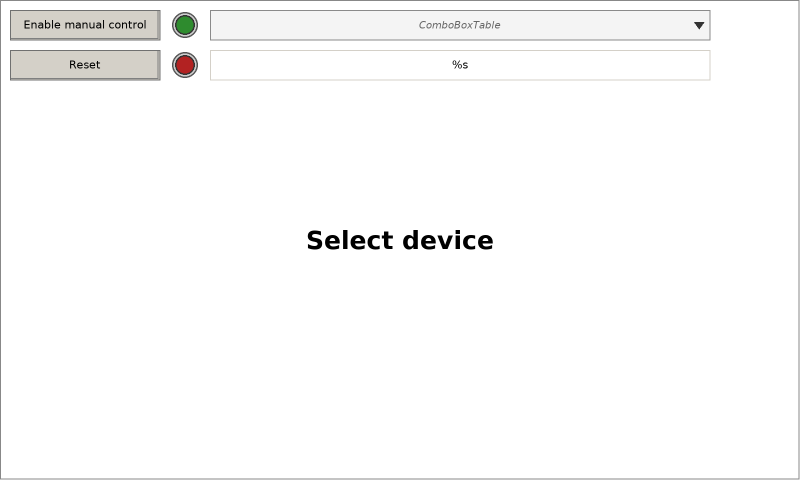
VISUALIZATION ManualControl  // 800x480
VAR_IN_OUT
	stHMI : UDT_HMI_ManualControl;
	fbManualController : FB_ManualController; // Only needed to reference the device array and its size
END_VAR
    Frame (0,0 800x480), input disabled if: NOT stHMI.bEnabled, frame switch variable: stHMI.refSelectedDevice.eDevType
        shows VisuUndefinedControl()
        shows VisuValveControl(pDev := stHMI.pDevValve)
        shows VisuCylinderControl(pDev := stHMI.pDevCylinder)
        shows VisuAxisControl(pDev := stHMI.pDevAxis)
        shows VisuPushbuttonLightControl(pDev := stHMI.pDevPBL)
        shows VisuDigitalInputControl(pDev := stHMI.pDevDigitalInput)
        shows VisuAnlogInputControl(pDev := stHMI.pDevAnalogInput)
        shows VisuDigitalOutControl(pDev := stHMI.pDevDigitalOut)
        shows VisuAnalogOutControl(pDev := stHMI.pDevAnalogOut)
        shows VisuPWMControl(pDev := stHMI.pDevPWMController)
        shows VisuDoublePWMControl(pDev := stHMI.pDevDoublePWM)
        shows VisuEncoderInput(pDev := stHMI.pDevEncoder)
        shows VisuAnalogAxisControl(pDev := stHMI.pDevAnalogAxis)
        shows VisuTwoVelocityAxisControl(pDev := stHMI.pDevTwoVelocityAxis)
        shows VisuKL5151Control(pDev := stHMI.pDevKL5151)
        shows VisuKL15XXControl(pDev := stHMI.pDevKL1512)
        pReferences[2]: HMI=stHMI
        pReferences[3]: HMI=stHMI
        pReferences[4]: HMI=stHMI
        pReferences[5]: HMI=stHMI
        pReferences[6]: HMI=stHMI
        pReferences[7]: HMI=stHMI
        pReferences[8]: HMI=stHMI
        pReferences[9]: HMI=stHMI
        pReferences[10]: HMI=stHMI
        pReferences[11]: HMI=stHMI
        pReferences[12]: HMI=stHMI
        pReferences[13]: HMI=stHMI
        pReferences[14]: HMI=stHMI
        pReferences[15]: HMI=stHMI
    Lamp1 (170,50 30x30), tooltip "component fault active", variable: stHMI.refSelectedDevice.bErrorActive, style: Lamp-Lamp1-Red
    Lamp1 (170,10 30x30), tooltip "Manual control active", variable: stHMI.bEnabled, style: Lamp-Lamp1-Green
    Textfield (210,50 500x30), "%s", text variable: stHMI.refSelectedDevice.sActiveState
    Button (10,50 150x30), "Reset", input disabled if: NOT stHMI.bEnabled
        tap stHMI.bReset
    ComboBoxTable (210,10 500x30), variable: stHMI.nSelectedDevice, data array: fbManualController.arDeviceArray
        p1128707560: fbManualController.nNumberOfDevices
        p3854506369: fbManualController.arDeviceArray[INDEX].sName
        p1892666644: fbManualController.arDeviceArray[INDEX].sType
        p338671338: fbManualController.arDeviceArray[INDEX].pFunction^
    Button (10,10 150x30), "Enable manual control", input disabled if: stHMI.bBlocked
        toggle stHMI.bEnabled
END_VISUALIZATION

// ---- _TESTS/VISU_TEST.TcVIS
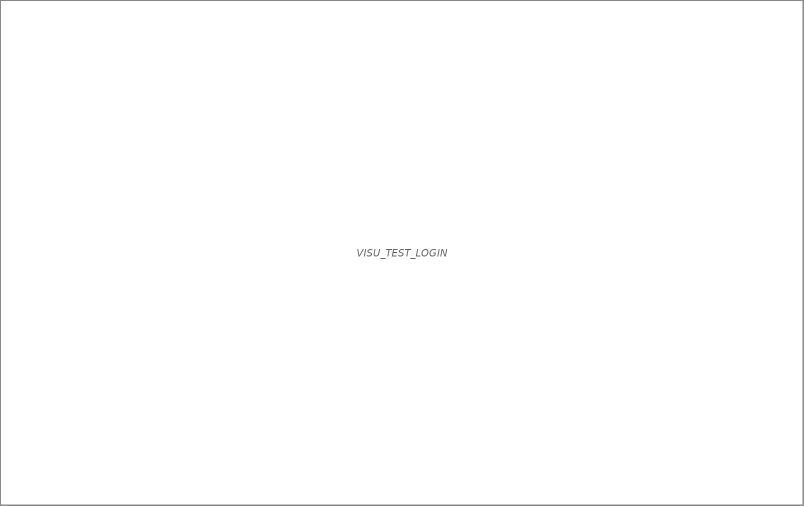
VISUALIZATION VISU_TEST  // 804x506
    TabControl (0,0 804x506)
        shows VISU_TEST_LOGIN()
        shows ManualControl(stHMI := PRG_TEST_FB_MANUALCONTROLLER.fbManualController.stHMI, fbManualController := PRG_TEST_FB_MANUALCONTROLLER.fbManualController)
        shows ParameterControl()
        [0]: TabTitle=Login
        [1]: TabTitle=ManualControl
        [2]: TabTitle=ParameterControl
END_VISUALIZATION

// ---- _TESTS/VISU_TEST_LOGIN.TcVIS
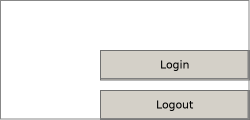
VISUALIZATION VISU_TEST_LOGIN  // 250x120
    Button (100,50 150x30), "Login"
        OnMouseDown: VisuUserMgmt Type=Login
    Button (100,90 150x30), "Logout"
        OnMouseDown: VisuUserMgmt Type=Logout
END_VISUALIZATION
